LIN {X 0,Y 516.781,Z 239.858,A -85,B 0,C 180,E1 -4940.608,E2 -4940.608} C_VEL
LIN {X 0,Y 516.85,Z 239.104,A -85,B 0,C 180,E1 -4941.398,E2 -4941.398} C_VEL
LIN {X 0,Y 517,Z 239.087,A -85,B 0,C 180,E1 -4943.757,E2 -4943.757} C_VEL
LIN {X 0,Y 517.072,Z 239.077,A -85,B 0,C 180,E1 -4947.663,E2 -4947.663} C_VEL
LIN {X 0,Y 517.085,Z 239.079,A -85,B 0,C 180,E1 -4950.779,E2 -4950.779} C_VEL
LIN {X 0,Y 517.006,Z 239.087,A -85,B 0,C 180,E1 -4953.117,E2 -4953.117} C_VEL
LIN {X 0,Y 517,Z 239.087,A -85,B 0,C 180,E1 -4956.243,E2 -4956.243} C_VEL
LIN {X 0,Y 516.949,Z 239.094,A -85,B 0,C 180,E1 -4959.389,E2 -4959.389} C_VEL
LIN {X 0,Y 516.972,Z 239.092,A -85,B 0,C 180,E1 -4961.824,E2 -4961.824} C_VEL
LIN {X 0,Y 516.933,Z 239.096,A -85,B 0,C 180,E1 -4965.147,E2 -4965.147} C_VEL
LIN {X 0,Y 516.915,Z 239.097,A -85,B 0,C 180,E1 -4968.222,E2 -4968.222} C_VEL
LIN {X 0,Y 516.904,Z 239.098,A -85,B 0,C 180,E1 -4970.702,E2 -4970.702} C_VEL
LIN {X 0,Y 516.881,Z 239.1,A -85,B 0,C 180,E1 -4973.223,E2 -4973.223} C_VEL
LIN {X 0,Y 516.934,Z 239.096,A -85,B 0,C 180,E1 -4976.197,E2 -4976.197} C_VEL
LIN {X 0,Y 516.925,Z 239.096,A -85,B 0,C 180,E1 -4979.304,E2 -4979.304} C_VEL
LIN {X 0,Y 516.889,Z 239.099,A -85,B 0,C 180,E1 -4982.545,E2 -4982.545} C_VEL
LIN {X 0,Y 516.871,Z 239.103,A -85,B 0,C 180,E1 -4985.333,E2 -4985.333} C_VEL
LIN {X 0,Y 516.871,Z 239.105,A -85,B 0,C 180,E1 -4987.944,E2 -4987.944} C_VEL
LIN {X 0,Y 516.893,Z 239.1,A -85,B 0,C 180,E1 -4990.74,E2 -4990.74} C_VEL
LIN {X 0,Y 516.872,Z 239.105,A -85,B 0,C 180,E1 -4993.903,E2 -4993.903} C_VEL
LIN {X 0,Y 516.872,Z 239.103,A -85,B 0,C 180,E1 -4996.107,E2 -4996.107} C_VEL
LIN {X 0,Y 516.893,Z 239.1,A -85,B 0,C 180,E1 -4999.261,E2 -4999.261} C_VEL
LIN {X 0,Y 516.871,Z 239.103,A -85,B 0,C 180,E1 -5002.057,E2 -5002.057} C_VEL
LIN {X 0,Y 516.884,Z 239.102,A -85,B 0,C 180,E1 -5005.177,E2 -5005.177} C_VEL
LIN {X 0,Y 516.872,Z 239.102,A -85,B 0,C 180,E1 -5007.976,E2 -5007.976} C_VEL
LIN {X 0,Y 516.926,Z 239.097,A -85,B 0,C 180,E1 -5010.697,E2 -5010.697} C_VEL
LIN {X 0,Y 516.935,Z 239.093,A -85,B 0,C 180,E1 -5013.804,E2 -5013.804} C_VEL
LIN {X 0,Y 516.862,Z 239.106,A -85,B 0,C 180,E1 -5016.777,E2 -5016.777} C_VEL
LIN {X 0,Y 516.93,Z 239.094,A -85,B 0,C 180,E1 -5019.732,E2 -5019.732} C_VEL
LIN {X 0,Y 516.922,Z 239.097,A -85,B 0,C 180,E1 -5022.597,E2 -5022.597} C_VEL
LIN {X 0,Y 516.933,Z 239.097,A -85,B 0,C 180,E1 -5025.031,E2 -5025.031} C_VEL
LIN {X 0,Y 516.957,Z 239.092,A -85,B 0,C 180,E1 -5028.235,E2 -5028.235} C_VEL
LIN {X 0,Y 516.964,Z 239.092,A -85,B 0,C 180,E1 -5031.401,E2 -5031.401} C_VEL
LIN {X 0,Y 517.002,Z 239.088,A -85,B 0,C 180,E1 -5033.758,E2 -5033.758} C_VEL
LIN {X 0,Y 517.077,Z 239.077,A -85,B 0,C 180,E1 -5037.664,E2 -5037.664} C_VEL
LIN {X 0,Y 517.089,Z 239.077,A -85,B 0,C 180,E1 -5040.78,E2 -5040.78} C_VEL
LIN {X 0,Y 517.008,Z 239.086,A -85,B 0,C 180,E1 -5043.118,E2 -5043.118} C_VEL
LIN {X 0,Y 517.003,Z 239.086,A -85,B 0,C 180,E1 -5046.244,E2 -5046.244} C_VEL
LIN {X 0,Y 516.947,Z 239.095,A -85,B 0,C 180,E1 -5049.39,E2 -5049.39} C_VEL
LIN {X 0,Y 516.978,Z 239.091,A -85,B 0,C 180,E1 -5051.825,E2 -5051.825} C_VEL
LIN {X 0,Y 516.939,Z 239.095,A -85,B 0,C 180,E1 -5055.147,E2 -5055.147} C_VEL
LIN {X 0,Y 516.921,Z 239.096,A -85,B 0,C 180,E1 -5058.223,E2 -5058.223} C_VEL
LIN {X 0,Y 516.908,Z 239.097,A -85,B 0,C 180,E1 -5060.702,E2 -5060.702} C_VEL
LIN {X 0,Y 516.908,Z 239.098,A -85,B 0,C 180,E1 -5064.073,E2 -5064.073} C_VEL
LIN {X 0,Y 516.923,Z 239.095,A -85,B 0,C 180,E1 -5066.659,E2 -5066.659} C_VEL
LIN {X 0,Y 516.908,Z 239.1,A -85,B 0,C 180,E1 -5069.525,E2 -5069.525} C_VEL
LIN {X 0,Y 516.891,Z 239.099,A -85,B 0,C 180,E1 -5072.544,E2 -5072.544} C_VEL
LIN {X 0,Y 516.878,Z 239.103,A -85,B 0,C 180,E1 -5075.333,E2 -5075.333} C_VEL
LIN {X 0,Y 516.88,Z 239.103,A -85,B 0,C 180,E1 -5077.944,E2 -5077.944} C_VEL
LIN {X 0,Y 516.883,Z 239.102,A -85,B 0,C 180,E1 -5080.742,E2 -5080.742} C_VEL
LIN {X 0,Y 516.882,Z 239.103,A -85,B 0,C 180,E1 -5082.832,E2 -5082.832} C_VEL
LIN {X 0,Y 516.895,Z 239.101,A -85,B 0,C 180,E1 -5085.008,E2 -5085.008} C_VEL
LIN {X 0,Y 516.917,Z 239.097,A -85,B 0,C 180,E1 -5088.399,E2 -5088.399} C_VEL
LIN {X 0,Y 516.883,Z 239.102,A -85,B 0,C 180,E1 -5091.285,E2 -5091.285} C_VEL
LIN {X 0,Y 516.887,Z 239.123,A -85,B 0,C 180,E1 -5092.277,E2 -5092.277} C_VEL
LIN {X 0,Y 517.553,Z 243.494,A -85,B 0,C 180,E1 -5094.275,E2 -5094.275} C_VEL
LIN {X 0,Y 517.476,Z 248.974,A -85,B 0,C 180,E1 -5096.631,E2 -5096.631} C_VEL
LIN {X 0,Y 517.259,Z 255.571,A -85,B 0,C 180,E1 -5099.369,E2 -5099.369} C_VEL
LIN {X 0,Y 517.082,Z 262.252,A -85,B 0,C 180,E1 -5102.063,E2 -5102.063} C_VEL
LIN {X 0,Y 516.871,Z 269.94,A -85,B 0,C 180,E1 -5105.07,E2 -5105.07} C_VEL
LIN {X 0,Y 516.754,Z 277.811,A -85,B 0,C 180,E1 -5108.046,E2 -5108.046} C_VEL
LIN {X 0,Y 516.65,Z 285.647,A -85,B 0,C 180,E1 -5110.945,E2 -5110.945} C_VEL
LIN {X 0,Y 516.556,Z 294.588,A -85,B 0,C 180,E1 -5114.21,E2 -5114.21} C_VEL
LIN {X 0,Y 516.475,Z 299.805,A -85,B 0,C 180,E1 -5116.098,E2 -5116.098} C_VEL
LIN {X 0,Y 518.444,Z 312.994,A -85,B 0,C 180,E1 -5116.477,E2 -5116.477} C_VEL
LIN {X 0,Y 518.159,Z 326.349,A -85,B 0,C 180,E1 -5116.968,E2 -5116.968} C_VEL
LIN {X 0,Y 517.84,Z 339.017,A -85,B 0,C 180,E1 -5117.611,E2 -5117.611} C_VEL
LIN {X 0,Y 517.528,Z 350.117,A -85,B 0,C 180,E1 -5118.346,E2 -5118.346} C_VEL
LIN {X 0,Y 517.27,Z 360.807,A -85,B 0,C 180,E1 -5119.233,E2 -5119.233} C_VEL
LIN {X 0,Y 516.954,Z 370.437,A -85,B 0,C 180,E1 -5120.216,E2 -5120.216} C_VEL
LIN {X 0,Y 516.748,Z 378.335,A -85,B 0,C 180,E1 -5121.199,E2 -5121.199} C_VEL
LIN {X 0,Y 516.557,Z 386.049,A -85,B 0,C 180,E1 -5122.377,E2 -5122.377} C_VEL
LIN {X 0,Y 516.41,Z 393.155,A -85,B 0,C 180,E1 -5123.75,E2 -5123.75} C_VEL
LIN {X 0,Y 516.313,Z 397.881,A -85,B 0,C 180,E1 -5124.924,E2 -5124.924} C_VEL
LIN {X 0,Y 516.353,Z 401.495,A -85,B 0,C 180,E1 -5126.098,E2 -5126.098} C_VEL
LIN {X 0,Y 516.283,Z 403.356,A -85,B 0,C 180,E1 -5126.879,E2 -5126.879} C_VEL
LIN {X 0,Y 516.262,Z 404.752,A -85,B 0,C 180,E1 -5127.659,E2 -5127.659} C_VEL
LIN {X 0,Y 516.16,Z 406.353,A -85,B 0,C 180,E1 -5129.22,E2 -5129.22} C_VEL
LIN {X 0,Y 516.154,Z 406.567,A -85,B 0,C 180,E1 -5130,E2 -5130} C_VEL
LIN {X 0,Y 516.192,Z 405.742,A -85,B 0,C 180,E1 -5131.56,E2 -5131.56} C_VEL
LIN {X 0,Y 516.262,Z 404.747,A -85,B 0,C 180,E1 -5132.34,E2 -5132.34} C_VEL
LIN {X 0,Y 516.283,Z 403.347,A -85,B 0,C 180,E1 -5133.121,E2 -5133.121} C_VEL
LIN {X 0,Y 516.312,Z 400.405,A -85,B 0,C 180,E1 -5134.293,E2 -5134.293} C_VEL
LIN {X 0,Y 516.376,Z 396.423,A -85,B 0,C 180,E1 -5135.467,E2 -5135.467} C_VEL
LIN {X 0,Y 516.476,Z 390.537,A -85,B 0,C 180,E1 -5136.792,E2 -5136.792} C_VEL
LIN {X 0,Y 516.607,Z 383.603,A -85,B 0,C 180,E1 -5138.015,E2 -5138.015} C_VEL
LIN {X 0,Y 516.828,Z 375.295,A -85,B 0,C 180,E1 -5139.194,E2 -5139.194} C_VEL
LIN {X 0,Y 517.045,Z 366.775,A -85,B 0,C 180,E1 -5140.178,E2 -5140.178} C_VEL
LIN {X 0,Y 517.372,Z 356.252,A -85,B 0,C 180,E1 -5141.161,E2 -5141.161} C_VEL
LIN {X 0,Y 517.64,Z 345.343,A -85,B 0,C 180,E1 -5141.984,E2 -5141.984} C_VEL
LIN {X 0,Y 517.922,Z 334.436,A -85,B 0,C 180,E1 -5142.639,E2 -5142.639} C_VEL
LIN {X 0,Y 518.242,Z 322.713,A -85,B 0,C 180,E1 -5143.179,E2 -5143.179} C_VEL
LIN {X 0,Y 518.222,Z 311.055,A -85,B 0,C 180,E1 -5143.579,E2 -5143.579} C_VEL
LIN {X 0,Y 516.474,Z 299.644,A -85,B 0,C 180,E1 -5143.901,E2 -5143.901} C_VEL
LIN {X 0,Y 516.546,Z 290.986,A -85,B 0,C 180,E1 -5147.009,E2 -5147.009} C_VEL
LIN {X 0,Y 516.662,Z 282.256,A -85,B 0,C 180,E1 -5150.183,E2 -5150.183} C_VEL
LIN {X 0,Y 516.778,Z 274.076,A -85,B 0,C 180,E1 -5153.227,E2 -5153.227} C_VEL
LIN {X 0,Y 516.93,Z 266.37,A -85,B 0,C 180,E1 -5156.192,E2 -5156.192} C_VEL
LIN {X 0,Y 517.175,Z 257.911,A -85,B 0,C 180,E1 -5159.574,E2 -5159.574} C_VEL
LIN {X 0,Y 517.338,Z 252.096,A -85,B 0,C 180,E1 -5161.992,E2 -5161.992} C_VEL
LIN {X 0,Y 517.55,Z 245.678,A -85,B 0,C 180,E1 -5164.773,E2 -5164.773} C_VEL
LIN {X 0,Y 517.485,Z 242.522,A -85,B 0,C 180,E1 -5166.211,E2 -5166.211} C_VEL
LIN {X 0,Y 516.903,Z 239.1,A -85,B 0,C 180,E1 -5167.945,E2 -5167.945} C_VEL
LIN {X 0,Y 516.883,Z 239.103,A -85,B 0,C 180,E1 -5170.741,E2 -5170.741} C_VEL
LIN {X 0,Y 516.904,Z 239.099,A -85,B 0,C 180,E1 -5172.828,E2 -5172.828} C_VEL
LIN {X 0,Y 516.921,Z 239.097,A -85,B 0,C 180,E1 -5175.009,E2 -5175.009} C_VEL
LIN {X 0,Y 516.921,Z 239.099,A -85,B 0,C 180,E1 -5178.397,E2 -5178.397} C_VEL
LIN {X 0,Y 516.884,Z 239.103,A -85,B 0,C 180,E1 -5181.284,E2 -5181.284} C_VEL
LIN {X 0,Y 516.889,Z 239.101,A -85,B 0,C 180,E1 -5184.22,E2 -5184.22} C_VEL
LIN {X 0,Y 516.894,Z 239.101,A -85,B 0,C 180,E1 -5187.052,E2 -5187.052} C_VEL
LIN {X 0,Y 516.898,Z 239.101,A -85,B 0,C 180,E1 -5189.796,E2 -5189.796} C_VEL
LIN {X 0,Y 516.924,Z 239.096,A -85,B 0,C 180,E1 -5192.466,E2 -5192.466} C_VEL
LIN {X 0,Y 516.905,Z 239.1,A -85,B 0,C 180,E1 -5195.071,E2 -5195.071} C_VEL
LIN {X 0,Y 516.864,Z 239.104,A -85,B 0,C 180,E1 -5197.621,E2 -5197.621} C_VEL
LIN {X 0,Y 516.926,Z 239.098,A -85,B 0,C 180,E1 -5200.129,E2 -5200.129} C_VEL
LIN {X 0,Y 516.925,Z 239.096,A -85,B 0,C 180,E1 -5202.595,E2 -5202.595} C_VEL
LIN {X 0,Y 516.935,Z 239.096,A -85,B 0,C 180,E1 -5205.029,E2 -5205.029} C_VEL
LIN {X 0,Y 516.958,Z 239.094,A -85,B 0,C 180,E1 -5208.233,E2 -5208.233} C_VEL
LIN {X 0,Y 516.966,Z 239.093,A -85,B 0,C 180,E1 -5211.399,E2 -5211.399} C_VEL
LIN {X 0,Y 517.003,Z 239.087,A -85,B 0,C 180,E1 -5213.756,E2 -5213.756} C_VEL
LIN {X 0,Y 517.008,Z 239.086,A -85,B 0,C 180,E1 -5216.882,E2 -5216.882} C_VEL
LIN {X 0,Y 517.076,Z 239.078,A -85,B 0,C 180,E1 -5219.999,E2 -5219.999} C_VEL
LIN {X 0,Y 517.009,Z 239.087,A -85,B 0,C 180,E1 -5223.116,E2 -5223.116} C_VEL
LIN {X 0,Y 517.002,Z 239.087,A -85,B 0,C 180,E1 -5226.242,E2 -5226.242} C_VEL
LIN {X 0,Y 516.938,Z 239.096,A -85,B 0,C 180,E1 -5229.388,E2 -5229.388} C_VEL
LIN {X 0,Y 516.852,Z 239.109,A -85,B 0,C 180,E1 -5230.181,E2 -5230.181} C_VEL
LIN {X 0,Y 516.871,Z 239.697,A -85,B 0,C 180,E1 -5230.973,E2 -5230.973} C_VEL
LIN {X 0,Y 516.812,Z 243.273,A -85,B 0,C 180,E1 -5233.365,E2 -5233.365} C_VEL
LIN {X 0,Y 516.772,Z 246.951,A -85,B 0,C 180,E1 -5235.782,E2 -5235.782} C_VEL
LIN {X 0,Y 516.66,Z 250.764,A -85,B 0,C 180,E1 -5238.231,E2 -5238.231} C_VEL
LIN {X 0,Y 516.602,Z 254.676,A -85,B 0,C 180,E1 -5240.713,E2 -5240.713} C_VEL
LIN {X 0,Y 516.512,Z 258.727,A -85,B 0,C 180,E1 -5243.239,E2 -5243.239} C_VEL
LIN {X 0,Y 516.464,Z 263.377,A -85,B 0,C 180,E1 -5246.09,E2 -5246.09} C_VEL
LIN {X 0,Y 516.368,Z 267.257,A -85,B 0,C 180,E1 -5248.447,E2 -5248.447} C_VEL
LIN {X 0,Y 516.307,Z 271.751,A -85,B 0,C 180,E1 -5251.147,E2 -5251.147} C_VEL
LIN {X 0,Y 516.332,Z 273.494,A -85,B 0,C 180,E1 -5252.181,E2 -5252.181} C_VEL
LIN {X 0,Y 518.441,Z 284.959,A -85,B 0,C 180,E1 -5252.535,E2 -5252.535} C_VEL
LIN {X 0,Y 518.197,Z 298.137,A -85,B 0,C 180,E1 -5253.026,E2 -5253.026} C_VEL
LIN {X 0,Y 517.923,Z 309.971,A -85,B 0,C 180,E1 -5253.627,E2 -5253.627} C_VEL
LIN {X 0,Y 517.63,Z 321.625,A -85,B 0,C 180,E1 -5254.398,E2 -5254.398} C_VEL
LIN {X 0,Y 517.328,Z 331.516,A -85,B 0,C 180,E1 -5255.217,E2 -5255.217} C_VEL
LIN {X 0,Y 517.051,Z 341.592,A -85,B 0,C 180,E1 -5256.246,E2 -5256.246} C_VEL
LIN {X 0,Y 516.815,Z 349.52,A -85,B 0,C 180,E1 -5257.237,E2 -5257.237} C_VEL
LIN {X 0,Y 516.593,Z 357.769,A -85,B 0,C 180,E1 -5258.519,E2 -5258.519} C_VEL
LIN {X 0,Y 516.449,Z 364.091,A -85,B 0,C 180,E1 -5259.76,E2 -5259.76} C_VEL
LIN {X 0,Y 516.345,Z 369.595,A -85,B 0,C 180,E1 -5261.16,E2 -5261.16} C_VEL
LIN {X 0,Y 516.273,Z 372.805,A -85,B 0,C 180,E1 -5262.254,E2 -5262.254} C_VEL
LIN {X 0,Y 516.175,Z 375.193,A -85,B 0,C 180,E1 -5263.418,E2 -5263.418} C_VEL
LIN {X 0,Y 515.501,Z 376.253,A -85,B 0,C 180,E1 -5264.06,E2 -5264.06} C_VEL
LIN {X 0,Y 512.613,Z 377.313,A -85,B 0,C 180,E1 -5265.11,E2 -5265.11} C_VEL
LIN {X 0,Y 510.18,Z 377.672,A -85,B 0,C 180,E1 -5265.961,E2 -5265.961} C_VEL
LIN {X 0,Y 509.086,Z 377.559,A -85,B 0,C 180,E1 -5266.731,E2 -5266.731} C_VEL
LIN {X 0,Y 509.067,Z 377.457,A -85,B 0,C 180,E1 -5266.842,E2 -5266.842} C_VEL
LIN {X 0,Y 509.1,Z 376.219,A -85,B 0,C 180,E1 -5268.196,E2 -5268.196} C_VEL
LIN {X 0,Y 509.152,Z 373.756,A -85,B 0,C 180,E1 -5269.553,E2 -5269.553} C_VEL
LIN {X 0,Y 509.246,Z 369.376,A -85,B 0,C 180,E1 -5271.112,E2 -5271.112} C_VEL
LIN {X 0,Y 509.371,Z 365.032,A -85,B 0,C 180,E1 -5272.243,E2 -5272.243} C_VEL
LIN {X 0,Y 509.524,Z 358.201,A -85,B 0,C 180,E1 -5273.623,E2 -5273.623} C_VEL
LIN {X 0,Y 509.749,Z 350.466,A -85,B 0,C 180,E1 -5274.858,E2 -5274.858} C_VEL
LIN {X 0,Y 510.002,Z 342.168,A -85,B 0,C 180,E1 -5275.928,E2 -5275.928} C_VEL
LIN {X 0,Y 510.286,Z 333.086,A -85,B 0,C 180,E1 -5276.885,E2 -5276.885} C_VEL
LIN {X 0,Y 510.534,Z 322.887,A -85,B 0,C 180,E1 -5277.763,E2 -5277.763} C_VEL
LIN {X 0,Y 510.843,Z 311.745,A -85,B 0,C 180,E1 -5278.534,E2 -5278.534} C_VEL
LIN {X 0,Y 511.18,Z 300.598,A -85,B 0,C 180,E1 -5279.137,E2 -5279.137} C_VEL
LIN {X 0,Y 511.527,Z 287.847,A -85,B 0,C 180,E1 -5279.646,E2 -5279.646} C_VEL
LIN {X 0,Y 511.045,Z 282.976,A -85,B 0,C 180,E1 -5279.814,E2 -5279.814} C_VEL
LIN {X 0,Y 509.176,Z 273.536,A -85,B 0,C 180,E1 -5280.12,E2 -5280.12} C_VEL
LIN {X 0,Y 509.257,Z 268.829,A -85,B 0,C 180,E1 -5282.909,E2 -5282.909} C_VEL
LIN {X 0,Y 509.302,Z 264.37,A -85,B 0,C 180,E1 -5285.606,E2 -5285.606} C_VEL
LIN {X 0,Y 509.405,Z 260.256,A -85,B 0,C 180,E1 -5288.13,E2 -5288.13} C_VEL
LIN {X 0,Y 509.488,Z 256.157,A -85,B 0,C 180,E1 -5290.667,E2 -5290.667} C_VEL
LIN {X 0,Y 509.517,Z 252.195,A -85,B 0,C 180,E1 -5293.163,E2 -5293.163} C_VEL
LIN {X 0,Y 509.625,Z 248.325,A -85,B 0,C 180,E1 -5295.628,E2 -5295.628} C_VEL
LIN {X 0,Y 509.795,Z 243.32,A -85,B 0,C 180,E1 -5298.872,E2 -5298.872} C_VEL
LIN {X 0,Y 509.787,Z 239.984,A -85,B 0,C 180,E1 -5301.278,E2 -5301.278} C_VEL
LIN {X 0,Y 509.968,Z 239.963,A -85,B 0,C 180,E1 -5303.671,E2 -5303.671} C_VEL
LIN {X 0,Y 510.044,Z 239.952,A -85,B 0,C 180,E1 -5307.631,E2 -5307.631} C_VEL
LIN {X 0,Y 510.044,Z 239.953,A -85,B 0,C 180,E1 -5310,E2 -5310} C_VEL
LIN {X 0,Y 510.047,Z 239.953,A -85,B 0,C 180,E1 -5312.369,E2 -5312.369} C_VEL
LIN {X 0,Y 509.968,Z 239.963,A -85,B 0,C 180,E1 -5316.33,E2 -5316.33} C_VEL
LIN {X 0,Y 509.909,Z 239.97,A -85,B 0,C 180,E1 -5318.72,E2 -5318.72} C_VEL
LIN {X 0,Y 509.94,Z 239.967,A -85,B 0,C 180,E1 -5321.931,E2 -5321.931} C_VEL
LIN {X 0,Y 509.882,Z 239.974,A -85,B 0,C 180,E1 -5325.242,E2 -5325.242} C_VEL
LIN {X 0,Y 509.878,Z 239.974,A -85,B 0,C 180,E1 -5328.001,E2 -5328.001} C_VEL
LIN {X 0,Y 509.847,Z 239.978,A -85,B 0,C 180,E1 -5331.002,E2 -5331.002} C_VEL
LIN {X 0,Y 509.84,Z 239.98,A -85,B 0,C 180,E1 -5333.563,E2 -5333.563} C_VEL
LIN {X 0,Y 509.903,Z 239.97,A -85,B 0,C 180,E1 -5336.379,E2 -5336.379} C_VEL
LIN {X 0,Y 509.875,Z 239.973,A -85,B 0,C 180,E1 -5338.844,E2 -5338.844} C_VEL
LIN {X 0,Y 509.815,Z 239.982,A -85,B 0,C 180,E1 -5341.59,E2 -5341.59} C_VEL
LIN {X 0,Y 509.842,Z 239.979,A -85,B 0,C 180,E1 -5344.414,E2 -5344.414} C_VEL
LIN {X 0,Y 509.808,Z 239.983,A -85,B 0,C 180,E1 -5347.341,E2 -5347.341} C_VEL
LIN {X 0,Y 509.85,Z 239.978,A -85,B 0,C 180,E1 -5350.38,E2 -5350.38} C_VEL
LIN {X 0,Y 509.829,Z 239.981,A -85,B 0,C 180,E1 -5353.065,E2 -5353.065} C_VEL
LIN {X 0,Y 509.819,Z 239.981,A -85,B 0,C 180,E1 -5355.793,E2 -5355.793} C_VEL
LIN {X 0,Y 509.855,Z 239.976,A -85,B 0,C 180,E1 -5358.576,E2 -5358.576} C_VEL
LIN {X 0,Y 509.845,Z 239.977,A -85,B 0,C 180,E1 -5361.786,E2 -5361.786} C_VEL
LIN {X 0,Y 509.835,Z 239.979,A -85,B 0,C 180,E1 -5364.624,E2 -5364.624} C_VEL
LIN {X 0,Y 509.855,Z 239.977,A -85,B 0,C 180,E1 -5367.482,E2 -5367.482} C_VEL
LIN {X 0,Y 509.871,Z 239.973,A -85,B 0,C 180,E1 -5370.27,E2 -5370.27} C_VEL
LIN {X 0,Y 509.877,Z 239.975,A -85,B 0,C 180,E1 -5372.945,E2 -5372.945} C_VEL
LIN {X 0,Y 509.86,Z 239.977,A -85,B 0,C 180,E1 -5375.575,E2 -5375.575} C_VEL
LIN {X 0,Y 509.813,Z 239.983,A -85,B 0,C 180,E1 -5378.149,E2 -5378.149} C_VEL
LIN {X 0,Y 509.856,Z 239.978,A -85,B 0,C 180,E1 -5380.682,E2 -5380.682} C_VEL
LIN {X 0,Y 509.878,Z 239.973,A -85,B 0,C 180,E1 -5383.176,E2 -5383.176} C_VEL
LIN {X 0,Y 509.854,Z 239.976,A -85,B 0,C 180,E1 -5385.635,E2 -5385.635} C_VEL
LIN {X 0,Y 509.91,Z 239.971,A -85,B 0,C 180,E1 -5388.876,E2 -5388.876} C_VEL
LIN {X 0,Y 509.944,Z 239.965,A -85,B 0,C 180,E1 -5392.079,E2 -5392.079} C_VEL
LIN {X 0,Y 509.975,Z 239.962,A -85,B 0,C 180,E1 -5394.465,E2 -5394.465} C_VEL
LIN {X 0,Y 510.048,Z 239.953,A -85,B 0,C 180,E1 -5397.632,E2 -5397.632} C_VEL
LIN {X 0,Y 510.059,Z 239.952,A -85,B 0,C 180,E1 -5400.79,E2 -5400.79} C_VEL
LIN {X 0,Y 509.951,Z 239.965,A -85,B 0,C 180,E1 -5403.161,E2 -5403.161} C_VEL
LIN {X 0,Y 509.972,Z 239.962,A -85,B 0,C 180,E1 -5406.331,E2 -5406.331} C_VEL
LIN {X 0,Y 509.91,Z 239.969,A -85,B 0,C 180,E1 -5408.721,E2 -5408.721} C_VEL
LIN {X 0,Y 509.946,Z 239.966,A -85,B 0,C 180,E1 -5411.931,E2 -5411.931} C_VEL
LIN {X 0,Y 509.889,Z 239.974,A -85,B 0,C 180,E1 -5415.243,E2 -5415.243} C_VEL
LIN {X 0,Y 509.884,Z 239.973,A -85,B 0,C 180,E1 -5418.002,E2 -5418.002} C_VEL
LIN {X 0,Y 509.846,Z 239.977,A -85,B 0,C 180,E1 -5421.003,E2 -5421.003} C_VEL
LIN {X 0,Y 509.866,Z 239.975,A -85,B 0,C 180,E1 -5424.427,E2 -5424.427} C_VEL
LIN {X 0,Y 509.883,Z 239.973,A -85,B 0,C 180,E1 -5427.057,E2 -5427.057} C_VEL
LIN {X 0,Y 509.854,Z 239.978,A -85,B 0,C 180,E1 -5429.752,E2 -5429.752} C_VEL
LIN {X 0,Y 509.864,Z 239.975,A -85,B 0,C 180,E1 -5432.774,E2 -5432.774} C_VEL
LIN {X 0,Y 509.838,Z 239.981,A -85,B 0,C 180,E1 -5435.582,E2 -5435.582} C_VEL
LIN {X 0,Y 509.849,Z 239.977,A -85,B 0,C 180,E1 -5438.339,E2 -5438.339} C_VEL
LIN {X 0,Y 509.855,Z 239.978,A -85,B 0,C 180,E1 -5441.426,E2 -5441.426} C_VEL
LIN {X 0,Y 509.838,Z 239.978,A -85,B 0,C 180,E1 -5444.671,E2 -5444.671} C_VEL
LIN {X 0,Y 509.859,Z 239.976,A -85,B 0,C 180,E1 -5448.104,E2 -5448.104} C_VEL
LIN {X 0,Y 509.847,Z 239.977,A -85,B 0,C 180,E1 -5450.648,E2 -5450.648} C_VEL
LIN {X 0,Y 509.89,Z 240.142,A -85,B 0,C 180,E1 -5452.168,E2 -5452.168} C_VEL
LIN {X 0,Y 510.554,Z 244.774,A -85,B 0,C 180,E1 -5454.308,E2 -5454.308} C_VEL
LIN {X 0,Y 510.466,Z 250.003,A -85,B 0,C 180,E1 -5456.585,E2 -5456.585} C_VEL
LIN {X 0,Y 510.23,Z 256.59,A -85,B 0,C 180,E1 -5459.36,E2 -5459.36} C_VEL
LIN {X 0,Y 510.045,Z 263.199,A -85,B 0,C 180,E1 -5462.064,E2 -5462.064} C_VEL
LIN {X 0,Y 509.856,Z 269.825,A -85,B 0,C 180,E1 -5464.703,E2 -5464.703} C_VEL
LIN {X 0,Y 509.723,Z 277.003,A -85,B 0,C 180,E1 -5467.487,E2 -5467.487} C_VEL
LIN {X 0,Y 509.588,Z 285.451,A -85,B 0,C 180,E1 -5470.671,E2 -5470.671} C_VEL
LIN {X 0,Y 509.484,Z 294.395,A -85,B 0,C 180,E1 -5473.985,E2 -5473.985} C_VEL
LIN {X 0,Y 509.387,Z 299.615,A -85,B 0,C 180,E1 -5475.901,E2 -5475.901} C_VEL
LIN {X 0,Y 511.503,Z 313.527,A -85,B 0,C 180,E1 -5476.315,E2 -5476.315} C_VEL
LIN {X 0,Y 511.216,Z 326.109,A -85,B 0,C 180,E1 -5476.788,E2 -5476.788} C_VEL
LIN {X 0,Y 510.891,Z 338.842,A -85,B 0,C 180,E1 -5477.443,E2 -5477.443} C_VEL
LIN {X 0,Y 510.528,Z 349.891,A -85,B 0,C 180,E1 -5478.184,E2 -5478.184} C_VEL
LIN {X 0,Y 510.269,Z 360.585,A -85,B 0,C 180,E1 -5479.083,E2 -5479.083} C_VEL
LIN {X 0,Y 509.921,Z 370.219,A -85,B 0,C 180,E1 -5480.08,E2 -5480.08} C_VEL
LIN {X 0,Y 509.696,Z 378.122,A -85,B 0,C 180,E1 -5481.076,E2 -5481.076} C_VEL
LIN {X 0,Y 509.488,Z 385.841,A -85,B 0,C 180,E1 -5482.271,E2 -5482.271} C_VEL
LIN {X 0,Y 509.322,Z 392.077,A -85,B 0,C 180,E1 -5483.472,E2 -5483.472} C_VEL
LIN {X 0,Y 509.244,Z 397.679,A -85,B 0,C 180,E1 -5484.853,E2 -5484.853} C_VEL
LIN {X 0,Y 509.246,Z 401.294,A -85,B 0,C 180,E1 -5486.043,E2 -5486.043} C_VEL
LIN {X 0,Y 509.201,Z 403.157,A -85,B 0,C 180,E1 -5486.835,E2 -5486.835} C_VEL
LIN {X 0,Y 509.19,Z 404.554,A -85,B 0,C 180,E1 -5487.627,E2 -5487.627} C_VEL
LIN {X 0,Y 509.074,Z 406.154,A -85,B 0,C 180,E1 -5489.209,E2 -5489.209} C_VEL
LIN {X 0,Y 509.066,Z 406.368,A -85,B 0,C 180,E1 -5490,E2 -5490} C_VEL
LIN {X 0,Y 509.113,Z 405.541,A -85,B 0,C 180,E1 -5491.582,E2 -5491.582} C_VEL
LIN {X 0,Y 509.19,Z 404.543,A -85,B 0,C 180,E1 -5492.373,E2 -5492.373} C_VEL
LIN {X 0,Y 509.201,Z 403.142,A -85,B 0,C 180,E1 -5493.165,E2 -5493.165} C_VEL
LIN {X 0,Y 509.205,Z 400.196,A -85,B 0,C 180,E1 -5494.353,E2 -5494.353} C_VEL
LIN {X 0,Y 509.294,Z 396.21,A -85,B 0,C 180,E1 -5495.543,E2 -5495.543} C_VEL
LIN {X 0,Y 509.409,Z 390.179,A -85,B 0,C 180,E1 -5496.913,E2 -5496.913} C_VEL
LIN {X 0,Y 509.552,Z 383.376,A -85,B 0,C 180,E1 -5498.127,E2 -5498.127} C_VEL
LIN {X 0,Y 509.775,Z 375.061,A -85,B 0,C 180,E1 -5499.322,E2 -5499.322} C_VEL
LIN {X 0,Y 510.022,Z 366.533,A -85,B 0,C 180,E1 -5500.319,E2 -5500.319} C_VEL
LIN {X 0,Y 510.374,Z 356.002,A -85,B 0,C 180,E1 -5501.316,E2 -5501.316} C_VEL
LIN {X 0,Y 510.643,Z 345.085,A -85,B 0,C 180,E1 -5502.151,E2 -5502.151} C_VEL
LIN {X 0,Y 510.975,Z 334.171,A -85,B 0,C 180,E1 -5502.814,E2 -5502.814} C_VEL
LIN {X 0,Y 511.304,Z 322.434,A -85,B 0,C 180,E1 -5503.361,E2 -5503.361} C_VEL
LIN {X 0,Y 511.295,Z 311.683,A -85,B 0,C 180,E1 -5503.741,E2 -5503.741} C_VEL
LIN {X 0,Y 509.377,Z 299.421,A -85,B 0,C 180,E1 -5504.099,E2 -5504.099} C_VEL
LIN {X 0,Y 509.486,Z 290.761,A -85,B 0,C 180,E1 -5507.252,E2 -5507.252} C_VEL
LIN {X 0,Y 509.593,Z 282.525,A -85,B 0,C 180,E1 -5510.311,E2 -5510.311} C_VEL
LIN {X 0,Y 509.73,Z 275.073,A -85,B 0,C 180,E1 -5513.138,E2 -5513.138} C_VEL
LIN {X 0,Y 509.906,Z 266.783,A -85,B 0,C 180,E1 -5516.376,E2 -5516.376} C_VEL
LIN {X 0,Y 510.14,Z 258.414,A -85,B 0,C 180,E1 -5519.781,E2 -5519.781} C_VEL
LIN {X 0,Y 510.39,Z 251.18,A -85,B 0,C 180,E1 -5522.863,E2 -5522.863} C_VEL
LIN {X 0,Y 510.574,Z 244.858,A -85,B 0,C 180,E1 -5525.695,E2 -5525.695} C_VEL
LIN {X 0,Y 509.864,Z 239.978,A -85,B 0,C 180,E1 -5528.145,E2 -5528.145} C_VEL
LIN {X 0,Y 509.856,Z 239.979,A -85,B 0,C 180,E1 -5531.424,E2 -5531.424} C_VEL
LIN {X 0,Y 509.855,Z 239.978,A -85,B 0,C 180,E1 -5534.667,E2 -5534.667} C_VEL
LIN {X 0,Y 509.859,Z 239.977,A -85,B 0,C 180,E1 -5538.102,E2 -5538.102} C_VEL
LIN {X 0,Y 509.857,Z 239.98,A -85,B 0,C 180,E1 -5540.648,E2 -5540.648} C_VEL
LIN {X 0,Y 509.834,Z 239.982,A -85,B 0,C 180,E1 -5543.647,E2 -5543.647} C_VEL
LIN {X 0,Y 509.859,Z 239.978,A -85,B 0,C 180,E1 -5546.538,E2 -5546.538} C_VEL
LIN {X 0,Y 509.847,Z 239.978,A -85,B 0,C 180,E1 -5549.334,E2 -5549.334} C_VEL
LIN {X 0,Y 509.89,Z 239.973,A -85,B 0,C 180,E1 -5552.054,E2 -5552.054} C_VEL
LIN {X 0,Y 509.872,Z 239.976,A -85,B 0,C 180,E1 -5554.703,E2 -5554.703} C_VEL
LIN {X 0,Y 509.822,Z 239.981,A -85,B 0,C 180,E1 -5557.456,E2 -5557.456} C_VEL
LIN {X 0,Y 509.911,Z 239.971,A -85,B 0,C 180,E1 -5559.844,E2 -5559.844} C_VEL
LIN {X 0,Y 509.881,Z 239.976,A -85,B 0,C 180,E1 -5563.174,E2 -5563.174} C_VEL
LIN {X 0,Y 509.858,Z 239.977,A -85,B 0,C 180,E1 -5565.633,E2 -5565.633} C_VEL
LIN {X 0,Y 509.911,Z 239.97,A -85,B 0,C 180,E1 -5568.874,E2 -5568.874} C_VEL
LIN {X 0,Y 509.945,Z 239.966,A -85,B 0,C 180,E1 -5572.077,E2 -5572.077} C_VEL
LIN {X 0,Y 509.977,Z 239.963,A -85,B 0,C 180,E1 -5574.463,E2 -5574.463} C_VEL
LIN {X 0,Y 510.047,Z 239.955,A -85,B 0,C 180,E1 -5577.63,E2 -5577.63} C_VEL
LIN {X 0,Y 510.057,Z 239.953,A -85,B 0,C 180,E1 -5580.789,E2 -5580.789} C_VEL
LIN {X 0,Y 509.951,Z 239.966,A -85,B 0,C 180,E1 -5583.159,E2 -5583.159} C_VEL
LIN {X 0,Y 509.97,Z 239.963,A -85,B 0,C 180,E1 -5586.329,E2 -5586.329} C_VEL
LIN {X 0,Y 509.907,Z 239.973,A -85,B 0,C 180,E1 -5588.719,E2 -5588.719} C_VEL
LIN {X 0,Y 509.791,Z 239.989,A -85,B 0,C 180,E1 -5590.323,E2 -5590.323} C_VEL
LIN {X 0,Y 509.858,Z 242.042,A -85,B 0,C 180,E1 -5591.932,E2 -5591.932} C_VEL
LIN {X 0,Y 509.747,Z 246.901,A -85,B 0,C 180,E1 -5595.185,E2 -5595.185} C_VEL
LIN {X 0,Y 509.642,Z 251.084,A -85,B 0,C 180,E1 -5597.919,E2 -5597.919} C_VEL
LIN {X 0,Y 509.508,Z 255.884,A -85,B 0,C 180,E1 -5601.015,E2 -5601.015} C_VEL
LIN {X 0,Y 509.429,Z 259.988,A -85,B 0,C 180,E1 -5603.582,E2 -5603.582} C_VEL
LIN {X 0,Y 509.392,Z 264.302,A -85,B 0,C 180,E1 -5606.263,E2 -5606.263} C_VEL
LIN {X 0,Y 509.279,Z 268.575,A -85,B 0,C 180,E1 -5608.88,E2 -5608.88} C_VEL
LIN {X 0,Y 509.258,Z 273.702,A -85,B 0,C 180,E1 -5611.977,E2 -5611.977} C_VEL
LIN {X 0,Y 511.513,Z 286.226,A -85,B 0,C 180,E1 -5612.385,E2 -5612.385} C_VEL
LIN {X 0,Y 511.28,Z 298.858,A -85,B 0,C 180,E1 -5612.872,E2 -5612.872} C_VEL
LIN {X 0,Y 510.98,Z 310.801,A -85,B 0,C 180,E1 -5613.494,E2 -5613.494} C_VEL
LIN {X 0,Y 510.657,Z 322.087,A -85,B 0,C 180,E1 -5614.26,E2 -5614.26} C_VEL
LIN {X 0,Y 510.317,Z 333.282,A -85,B 0,C 180,E1 -5615.217,E2 -5615.217} C_VEL
LIN {X 0,Y 510.038,Z 342.078,A -85,B 0,C 180,E1 -5616.144,E2 -5616.144} C_VEL
LIN {X 0,Y 509.807,Z 349.558,A -85,B 0,C 180,E1 -5617.095,E2 -5617.095} C_VEL
LIN {X 0,Y 509.553,Z 357.672,A -85,B 0,C 180,E1 -5618.363,E2 -5618.363} C_VEL
LIN {X 0,Y 509.393,Z 364.178,A -85,B 0,C 180,E1 -5619.648,E2 -5619.648} C_VEL
LIN {X 0,Y 509.27,Z 369.573,A -85,B 0,C 180,E1 -5621.025,E2 -5621.025} C_VEL
LIN {X 0,Y 509.23,Z 371.983,A -85,B 0,C 180,E1 -5621.819,E2 -5621.819} C_VEL
LIN {X 0,Y 509.11,Z 374.729,A -85,B 0,C 180,E1 -5622.977,E2 -5622.977} C_VEL
LIN {X 0,Y 509.1,Z 376.556,A -85,B 0,C 180,E1 -5624.124,E2 -5624.124} C_VEL
LIN {X 0,Y 509.102,Z 377.498,A -85,B 0,C 180,E1 -5625.249,E2 -5625.249} C_VEL
LIN {X 0,Y 509.077,Z 377.658,A -85,B 0,C 180,E1 -5626.35,E2 -5626.35} C_VEL
LIN {X 0,Y 509.067,Z 377.457,A -85,B 0,C 180,E1 -5626.842,E2 -5626.842} C_VEL
LIN {X 0,Y 508.416,Z 377.061,A -85,B 0,C 180,E1 -5627.502,E2 -5627.502} C_VEL
LIN {X 0,Y 505.578,Z 375.823,A -85,B 0,C 180,E1 -5628.567,E2 -5628.567} C_VEL
LIN {X 0,Y 503.187,Z 374.316,A -85,B 0,C 180,E1 -5629.416,E2 -5629.416} C_VEL
LIN {X 0,Y 502.178,Z 372.853,A -85,B 0,C 180,E1 -5630.062,E2 -5630.062} C_VEL
LIN {X 0,Y 502.107,Z 372.281,A -85,B 0,C 180,E1 -5630.279,E2 -5630.279} C_VEL
LIN {X 0,Y 502.217,Z 368.114,A -85,B 0,C 180,E1 -5631.595,E2 -5631.595} C_VEL
LIN {X 0,Y 502.365,Z 362.072,A -85,B 0,C 180,E1 -5633.019,E2 -5633.019} C_VEL
LIN {X 0,Y 502.591,Z 354.402,A -85,B 0,C 180,E1 -5634.409,E2 -5634.409} C_VEL
LIN {X 0,Y 502.843,Z 346.536,A -85,B 0,C 180,E1 -5635.547,E2 -5635.547} C_VEL
LIN {X 0,Y 503.172,Z 337.297,A -85,B 0,C 180,E1 -5636.627,E2 -5636.627} C_VEL
LIN {X 0,Y 503.479,Z 326.916,A -85,B 0,C 180,E1 -5637.611,E2 -5637.611} C_VEL
LIN {X 0,Y 503.81,Z 316.676,A -85,B 0,C 180,E1 -5638.396,E2 -5638.396} C_VEL
LIN {X 0,Y 504.08,Z 305.816,A -85,B 0,C 180,E1 -5639.062,E2 -5639.062} C_VEL
LIN {X 0,Y 504.499,Z 293.122,A -85,B 0,C 180,E1 -5639.648,E2 -5639.648} C_VEL
LIN {X 0,Y 504.471,Z 285.768,A -85,B 0,C 180,E1 -5639.916,E2 -5639.916} C_VEL
LIN {X 0,Y 502.095,Z 273.703,A -85,B 0,C 180,E1 -5640.32,E2 -5640.32} C_VEL
LIN {X 0,Y 502.188,Z 268.596,A -85,B 0,C 180,E1 -5643.396,E2 -5643.396} C_VEL
LIN {X 0,Y 502.238,Z 264.247,A -85,B 0,C 180,E1 -5646.059,E2 -5646.059} C_VEL
LIN {X 0,Y 502.347,Z 260.031,A -85,B 0,C 180,E1 -5648.67,E2 -5648.67} C_VEL
LIN {X 0,Y 502.421,Z 255.955,A -85,B 0,C 180,E1 -5651.233,E2 -5651.233} C_VEL
LIN {X 0,Y 502.51,Z 250.7,A -85,B 0,C 180,E1 -5654.59,E2 -5654.59} C_VEL
LIN {X 0,Y 502.693,Z 245.617,A -85,B 0,C 180,E1 -5657.895,E2 -5657.895} C_VEL
LIN {X 0,Y 502.717,Z 240.866,A -85,B 0,C 180,E1 -5661.154,E2 -5661.154} C_VEL
LIN {X 0,Y 502.915,Z 240.842,A -85,B 0,C 180,E1 -5663.581,E2 -5663.581} C_VEL
LIN {X 0,Y 502.891,Z 240.845,A -85,B 0,C 180,E1 -5666.796,E2 -5666.796} C_VEL
LIN {X 0,Y 503.027,Z 240.827,A -85,B 0,C 180,E1 -5669.2,E2 -5669.2} C_VEL
LIN {X 0,Y 503.017,Z 240.829,A -85,B 0,C 180,E1 -5672.402,E2 -5672.402} C_VEL
LIN {X 0,Y 502.929,Z 240.84,A -85,B 0,C 180,E1 -5675.614,E2 -5675.614} C_VEL
LIN {X 0,Y 502.892,Z 240.846,A -85,B 0,C 180,E1 -5678.033,E2 -5678.033} C_VEL
LIN {X 0,Y 502.884,Z 240.844,A -85,B 0,C 180,E1 -5681.283,E2 -5681.283} C_VEL
LIN {X 0,Y 502.834,Z 240.851,A -85,B 0,C 180,E1 -5684.571,E2 -5684.571} C_VEL
LIN {X 0,Y 502.851,Z 240.85,A -85,B 0,C 180,E1 -5687.907,E2 -5687.907} C_VEL
LIN {X 0,Y 502.819,Z 240.852,A -85,B 0,C 180,E1 -5690.537,E2 -5690.537} C_VEL
LIN {X 0,Y 502.795,Z 240.854,A -85,B 0,C 180,E1 -5693.04,E2 -5693.04} C_VEL
LIN {X 0,Y 502.831,Z 240.852,A -85,B 0,C 180,E1 -5695.676,E2 -5695.676} C_VEL
LIN {X 0,Y 502.831,Z 240.853,A -85,B 0,C 180,E1 -5698.373,E2 -5698.373} C_VEL
LIN {X 0,Y 502.786,Z 240.857,A -85,B 0,C 180,E1 -5701.5,E2 -5701.5} C_VEL
LIN {X 0,Y 502.795,Z 240.857,A -85,B 0,C 180,E1 -5704.445,E2 -5704.445} C_VEL
LIN {X 0,Y 502.77,Z 240.86,A -85,B 0,C 180,E1 -5707.179,E2 -5707.179} C_VEL
LIN {X 0,Y 502.815,Z 240.854,A -85,B 0,C 180,E1 -5710.012,E2 -5710.012} C_VEL
LIN {X 0,Y 502.818,Z 240.852,A -85,B 0,C 180,E1 -5712.203,E2 -5712.203} C_VEL
LIN {X 0,Y 502.789,Z 240.858,A -85,B 0,C 180,E1 -5715.469,E2 -5715.469} C_VEL
LIN {X 0,Y 502.818,Z 240.853,A -85,B 0,C 180,E1 -5717.865,E2 -5717.865} C_VEL
LIN {X 0,Y 502.81,Z 240.855,A -85,B 0,C 180,E1 -5721.026,E2 -5721.026} C_VEL
LIN {X 0,Y 502.775,Z 240.857,A -85,B 0,C 180,E1 -5724.168,E2 -5724.168} C_VEL
LIN {X 0,Y 502.822,Z 240.854,A -85,B 0,C 180,E1 -5726.994,E2 -5726.994} C_VEL
LIN {X 0,Y 502.82,Z 240.852,A -85,B 0,C 180,E1 -5730.062,E2 -5730.062} C_VEL
LIN {X 0,Y 502.825,Z 240.852,A -85,B 0,C 180,E1 -5732.534,E2 -5732.534} C_VEL
LIN {X 0,Y 502.819,Z 240.854,A -85,B 0,C 180,E1 -5735.299,E2 -5735.299} C_VEL
LIN {X 0,Y 502.775,Z 240.859,A -85,B 0,C 180,E1 -5737.827,E2 -5737.827} C_VEL
LIN {X 0,Y 502.817,Z 240.855,A -85,B 0,C 180,E1 -5740.401,E2 -5740.401} C_VEL
LIN {X 0,Y 502.827,Z 240.853,A -85,B 0,C 180,E1 -5742.933,E2 -5742.933} C_VEL
LIN {X 0,Y 502.836,Z 240.851,A -85,B 0,C 180,E1 -5745.43,E2 -5745.43} C_VEL
LIN {X 0,Y 502.873,Z 240.849,A -85,B 0,C 180,E1 -5748.718,E2 -5748.718} C_VEL
LIN {X 0,Y 502.895,Z 240.843,A -85,B 0,C 180,E1 -5751.968,E2 -5751.968} C_VEL
LIN {X 0,Y 502.931,Z 240.839,A -85,B 0,C 180,E1 -5754.387,E2 -5754.387} C_VEL
LIN {X 0,Y 503.018,Z 240.828,A -85,B 0,C 180,E1 -5757.599,E2 -5757.599} C_VEL
LIN {X 0,Y 503.018,Z 240.829,A -85,B 0,C 180,E1 -5760.001,E2 -5760.001} C_VEL
LIN {X 0,Y 503.019,Z 240.828,A -85,B 0,C 180,E1 -5762.403,E2 -5762.403} C_VEL
LIN {X 0,Y 502.932,Z 240.84,A -85,B 0,C 180,E1 -5765.614,E2 -5765.614} C_VEL
LIN {X 0,Y 502.896,Z 240.846,A -85,B 0,C 180,E1 -5768.034,E2 -5768.034} C_VEL
LIN {X 0,Y 502.887,Z 240.843,A -85,B 0,C 180,E1 -5771.284,E2 -5771.284} C_VEL
LIN {X 0,Y 502.84,Z 240.849,A -85,B 0,C 180,E1 -5774.572,E2 -5774.572} C_VEL
LIN {X 0,Y 502.857,Z 240.849,A -85,B 0,C 180,E1 -5777.908,E2 -5777.908} C_VEL
LIN {X 0,Y 502.825,Z 240.851,A -85,B 0,C 180,E1 -5780.537,E2 -5780.537} C_VEL
LIN {X 0,Y 502.791,Z 240.856,A -85,B 0,C 180,E1 -5783.041,E2 -5783.041} C_VEL
LIN {X 0,Y 502.837,Z 240.852,A -85,B 0,C 180,E1 -5785.677,E2 -5785.677} C_VEL
LIN {X 0,Y 502.838,Z 240.851,A -85,B 0,C 180,E1 -5788.374,E2 -5788.374} C_VEL
LIN {X 0,Y 502.79,Z 240.857,A -85,B 0,C 180,E1 -5791.5,E2 -5791.5} C_VEL
LIN {X 0,Y 502.79,Z 240.857,A -85,B 0,C 180,E1 -5793.996,E2 -5793.996} C_VEL
LIN {X 0,Y 502.779,Z 240.859,A -85,B 0,C 180,E1 -5797.179,E2 -5797.179} C_VEL
LIN {X 0,Y 502.787,Z 240.857,A -85,B 0,C 180,E1 -5800.016,E2 -5800.016} C_VEL
LIN {X 0,Y 502.802,Z 240.853,A -85,B 0,C 180,E1 -5802.2,E2 -5802.2} C_VEL
LIN {X 0,Y 502.785,Z 240.857,A -85,B 0,C 180,E1 -5805.471,E2 -5805.471} C_VEL
LIN {X 0,Y 502.821,Z 240.854,A -85,B 0,C 180,E1 -5808.935,E2 -5808.935} C_VEL
LIN {X 0,Y 502.815,Z 240.872,A -85,B 0,C 180,E1 -5811.916,E2 -5811.916} C_VEL
LIN {X 0,Y 503.523,Z 245.535,A -85,B 0,C 180,E1 -5814.111,E2 -5814.111} C_VEL
LIN {X 0,Y 503.517,Z 249.912,A -85,B 0,C 180,E1 -5816.061,E2 -5816.061} C_VEL
LIN {X 0,Y 503.255,Z 256.495,A -85,B 0,C 180,E1 -5818.889,E2 -5818.889} C_VEL
LIN {X 0,Y 503.032,Z 263.163,A -85,B 0,C 180,E1 -5821.666,E2 -5821.666} C_VEL
LIN {X 0,Y 502.816,Z 270.837,A -85,B 0,C 180,E1 -5824.767,E2 -5824.767} C_VEL
LIN {X 0,Y 502.636,Z 278.578,A -85,B 0,C 180,E1 -5827.82,E2 -5827.82} C_VEL
LIN {X 0,Y 502.517,Z 286.378,A -85,B 0,C 180,E1 -5830.813,E2 -5830.813} C_VEL
LIN {X 0,Y 502.39,Z 295.317,A -85,B 0,C 180,E1 -5834.17,E2 -5834.17} C_VEL
LIN {X 0,Y 502.304,Z 299.424,A -85,B 0,C 180,E1 -5835.698,E2 -5835.698} C_VEL
LIN {X 0,Y 504.586,Z 314.05,A -85,B 0,C 180,E1 -5836.15,E2 -5836.15} C_VEL
LIN {X 0,Y 504.279,Z 326.993,A -85,B 0,C 180,E1 -5836.654,E2 -5836.654} C_VEL
LIN {X 0,Y 503.926,Z 338.902,A -85,B 0,C 180,E1 -5837.284,E2 -5837.284} C_VEL
LIN {X 0,Y 503.541,Z 349.664,A -85,B 0,C 180,E1 -5838.018,E2 -5838.018} C_VEL
LIN {X 0,Y 503.27,Z 360.363,A -85,B 0,C 180,E1 -5838.93,E2 -5838.93} C_VEL
LIN {X 0,Y 502.874,Z 370.001,A -85,B 0,C 180,E1 -5839.939,E2 -5839.939} C_VEL
LIN {X 0,Y 502.66,Z 377.909,A -85,B 0,C 180,E1 -5840.95,E2 -5840.95} C_VEL
LIN {X 0,Y 502.41,Z 385.632,A -85,B 0,C 180,E1 -5842.161,E2 -5842.161} C_VEL
LIN {X 0,Y 502.238,Z 392.335,A -85,B 0,C 180,E1 -5843.482,E2 -5843.482} C_VEL
LIN {X 0,Y 502.175,Z 397.477,A -85,B 0,C 180,E1 -5844.781,E2 -5844.781} C_VEL
LIN {X 0,Y 502.139,Z 401.093,A -85,B 0,C 180,E1 -5845.987,E2 -5845.987} C_VEL
LIN {X 0,Y 502.121,Z 402.958,A -85,B 0,C 180,E1 -5846.79,E2 -5846.79} C_VEL
LIN {X 0,Y 502.092,Z 404.355,A -85,B 0,C 180,E1 -5847.593,E2 -5847.593} C_VEL
LIN {X 0,Y 501.991,Z 405.955,A -85,B 0,C 180,E1 -5849.198,E2 -5849.198} C_VEL
LIN {X 0,Y 501.98,Z 406.169,A -85,B 0,C 180,E1 -5850,E2 -5850} C_VEL
LIN {X 0,Y 502.037,Z 405.34,A -85,B 0,C 180,E1 -5851.604,E2 -5851.604} C_VEL
LIN {X 0,Y 502.092,Z 404.34,A -85,B 0,C 180,E1 -5852.407,E2 -5852.407} C_VEL
LIN {X 0,Y 502.121,Z 402.936,A -85,B 0,C 180,E1 -5853.209,E2 -5853.209} C_VEL
LIN {X 0,Y 502.103,Z 399.986,A -85,B 0,C 180,E1 -5854.415,E2 -5854.415} C_VEL
LIN {X 0,Y 502.212,Z 395.996,A -85,B 0,C 180,E1 -5855.621,E2 -5855.621} C_VEL
LIN {X 0,Y 502.334,Z 389.959,A -85,B 0,C 180,E1 -5857.011,E2 -5857.011} C_VEL
LIN {X 0,Y 502.483,Z 383.149,A -85,B 0,C 180,E1 -5858.242,E2 -5858.242} C_VEL
LIN {X 0,Y 502.736,Z 374.827,A -85,B 0,C 180,E1 -5859.454,E2 -5859.454} C_VEL
LIN {X 0,Y 503.002,Z 366.291,A -85,B 0,C 180,E1 -5860.465,E2 -5860.465} C_VEL
LIN {X 0,Y 503.381,Z 355.751,A -85,B 0,C 180,E1 -5861.475,E2 -5861.475} C_VEL
LIN {X 0,Y 503.663,Z 344.828,A -85,B 0,C 180,E1 -5862.322,E2 -5862.322} C_VEL
LIN {X 0,Y 504.052,Z 333.907,A -85,B 0,C 180,E1 -5862.993,E2 -5862.993} C_VEL
LIN {X 0,Y 504.395,Z 322.157,A -85,B 0,C 180,E1 -5863.547,E2 -5863.547} C_VEL
LIN {X 0,Y 504.343,Z 312.281,A -85,B 0,C 180,E1 -5863.908,E2 -5863.908} C_VEL
LIN {X 0,Y 502.292,Z 299.198,A -85,B 0,C 180,E1 -5864.302,E2 -5864.302} C_VEL
LIN {X 0,Y 502.407,Z 290.566,A -85,B 0,C 180,E1 -5867.503,E2 -5867.503} C_VEL
LIN {X 0,Y 502.546,Z 282.736,A -85,B 0,C 180,E1 -5870.464,E2 -5870.464} C_VEL
LIN {X 0,Y 502.659,Z 274.922,A -85,B 0,C 180,E1 -5873.482,E2 -5873.482} C_VEL
LIN {X 0,Y 502.844,Z 268.301,A -85,B 0,C 180,E1 -5876.117,E2 -5876.117} C_VEL
LIN {X 0,Y 503.116,Z 260.638,A -85,B 0,C 180,E1 -5879.268,E2 -5879.268} C_VEL
LIN {X 0,Y 503.35,Z 253.088,A -85,B 0,C 180,E1 -5882.516,E2 -5882.516} C_VEL
LIN {X 0,Y 503.586,Z 246.725,A -85,B 0,C 180,E1 -5885.391,E2 -5885.391} C_VEL
LIN {X 0,Y 503.185,Z 242.946,A -85,B 0,C 180,E1 -5887.238,E2 -5887.238} C_VEL
LIN {X 0,Y 502.814,Z 240.856,A -85,B 0,C 180,E1 -5888.364,E2 -5888.364} C_VEL
LIN {X 0,Y 502.819,Z 240.855,A -85,B 0,C 180,E1 -5891.065,E2 -5891.065} C_VEL
LIN {X 0,Y 502.781,Z 240.861,A -85,B 0,C 180,E1 -5893.375,E2 -5893.375} C_VEL
LIN {X 0,Y 502.789,Z 240.859,A -85,B 0,C 180,E1 -5895.66,E2 -5895.66} C_VEL
LIN {X 0,Y 502.825,Z 240.854,A -85,B 0,C 180,E1 -5899.003,E2 -5899.003} C_VEL
LIN {X 0,Y 502.794,Z 240.857,A -85,B 0,C 180,E1 -5902.045,E2 -5902.045} C_VEL
LIN {X 0,Y 502.807,Z 240.855,A -85,B 0,C 180,E1 -5905.034,E2 -5905.034} C_VEL
LIN {X 0,Y 502.784,Z 240.859,A -85,B 0,C 180,E1 -5907.915,E2 -5907.915} C_VEL
LIN {X 0,Y 502.835,Z 240.853,A -85,B 0,C 180,E1 -5910.712,E2 -5910.712} C_VEL
LIN {X 0,Y 502.858,Z 240.848,A -85,B 0,C 180,E1 -5913.438,E2 -5913.438} C_VEL
LIN {X 0,Y 502.786,Z 240.859,A -85,B 0,C 180,E1 -5916.085,E2 -5916.085} C_VEL
LIN {X 0,Y 502.778,Z 240.859,A -85,B 0,C 180,E1 -5918.688,E2 -5918.688} C_VEL
LIN {X 0,Y 502.825,Z 240.854,A -85,B 0,C 180,E1 -5921.247,E2 -5921.247} C_VEL
LIN {X 0,Y 502.817,Z 240.854,A -85,B 0,C 180,E1 -5923.766,E2 -5923.766} C_VEL
LIN {X 0,Y 502.825,Z 240.854,A -85,B 0,C 180,E1 -5926.254,E2 -5926.254} C_VEL
LIN {X 0,Y 502.875,Z 240.846,A -85,B 0,C 180,E1 -5928.716,E2 -5928.716} C_VEL
LIN {X 0,Y 502.895,Z 240.844,A -85,B 0,C 180,E1 -5931.966,E2 -5931.966} C_VEL
LIN {X 0,Y 502.932,Z 240.841,A -85,B 0,C 180,E1 -5934.386,E2 -5934.386} C_VEL
LIN {X 0,Y 503.017,Z 240.831,A -85,B 0,C 180,E1 -5937.597,E2 -5937.597} C_VEL
LIN {X 0,Y 503.018,Z 240.829,A -85,B 0,C 180,E1 -5939.999,E2 -5939.999} C_VEL
LIN {X 0,Y 503.018,Z 240.83,A -85,B 0,C 180,E1 -5942.401,E2 -5942.401} C_VEL
LIN {X 0,Y 502.931,Z 240.841,A -85,B 0,C 180,E1 -5945.613,E2 -5945.613} C_VEL
LIN {X 0,Y 502.892,Z 240.846,A -85,B 0,C 180,E1 -5948.032,E2 -5948.032} C_VEL
LIN {X 0,Y 502.737,Z 240.89,A -85,B 0,C 180,E1 -5950.47,E2 -5950.47} C_VEL
LIN {X 0,Y 502.762,Z 244.424,A -85,B 0,C 180,E1 -5952.923,E2 -5952.923} C_VEL
LIN {X 0,Y 502.683,Z 248.093,A -85,B 0,C 180,E1 -5955.404,E2 -5955.404} C_VEL
LIN {X 0,Y 502.578,Z 252.062,A -85,B 0,C 180,E1 -5958.032,E2 -5958.032} C_VEL
LIN {X 0,Y 502.446,Z 257.131,A -85,B 0,C 180,E1 -5961.325,E2 -5961.325} C_VEL
LIN {X 0,Y 502.344,Z 261.23,A -85,B 0,C 180,E1 -5963.935,E2 -5963.935} C_VEL
LIN {X 0,Y 502.293,Z 265.483,A -85,B 0,C 180,E1 -5966.597,E2 -5966.597} C_VEL
LIN {X 0,Y 502.184,Z 269.912,A -85,B 0,C 180,E1 -5969.327,E2 -5969.327} C_VEL
LIN {X 0,Y 502.195,Z 274.071,A -85,B 0,C 180,E1 -5971.794,E2 -5971.794} C_VEL
LIN {X 0,Y 504.573,Z 286.303,A -85,B 0,C 180,E1 -5972.191,E2 -5972.191} C_VEL
LIN {X 0,Y 504.382,Z 298.775,A -85,B 0,C 180,E1 -5972.678,E2 -5972.678} C_VEL
LIN {X 0,Y 504.039,Z 311.083,A -85,B 0,C 180,E1 -5973.326,E2 -5973.326} C_VEL
LIN {X 0,Y 503.669,Z 322.892,A -85,B 0,C 180,E1 -5974.144,E2 -5974.144} C_VEL
LIN {X 0,Y 503.343,Z 333.229,A -85,B 0,C 180,E1 -5975.043,E2 -5975.043} C_VEL
LIN {X 0,Y 503.009,Z 342.686,A -85,B 0,C 180,E1 -5976.054,E2 -5976.054} C_VEL
LIN {X 0,Y 502.732,Z 351.148,A -85,B 0,C 180,E1 -5977.172,E2 -5977.172} C_VEL
LIN {X 0,Y 502.483,Z 358.901,A -85,B 0,C 180,E1 -5978.443,E2 -5978.443} C_VEL
LIN {X 0,Y 502.307,Z 364.963,A -85,B 0,C 180,E1 -5979.69,E2 -5979.69} C_VEL
LIN {X 0,Y 502.193,Z 370.313,A -85,B 0,C 180,E1 -5981.127,E2 -5981.127} C_VEL
LIN {X 0,Y 502.089,Z 373.365,A -85,B 0,C 180,E1 -5982.211,E2 -5982.211} C_VEL
LIN {X 0,Y 501.999,Z 375.608,A -85,B 0,C 180,E1 -5983.313,E2 -5983.313} C_VEL
LIN {X 0,Y 502.025,Z 377.106,A -85,B 0,C 180,E1 -5984.443,E2 -5984.443} C_VEL
LIN {X 0,Y 501.998,Z 377.828,A -85,B 0,C 180,E1 -5985.574,E2 -5985.574} C_VEL
LIN {X 0,Y 501.972,Z 377.678,A -85,B 0,C 180,E1 -5986.839,E2 -5986.839} C_VEL
LIN {X 0,Y 501.99,Z 376.838,A -85,B 0,C 180,E1 -5987.901,E2 -5987.901} C_VEL
LIN {X 0,Y 502.049,Z 374.991,A -85,B 0,C 180,E1 -5989.104,E2 -5989.104} C_VEL
LIN {X 0,Y 502.107,Z 372.281,A -85,B 0,C 180,E1 -5990.279,E2 -5990.279} C_VEL
LIN {X 0,Y 501.484,Z 370.49,A -85,B 0,C 180,E1 -5990.919,E2 -5990.919} C_VEL
LIN {X 0,Y 498.715,Z 367.13,A -85,B 0,C 180,E1 -5991.941,E2 -5991.941} C_VEL
LIN {X 0,Y 495.965,Z 363.071,A -85,B 0,C 180,E1 -5992.938,E2 -5992.938} C_VEL
LIN {X 0,Y 495.379,Z 360.184,A -85,B 0,C 180,E1 -5993.533,E2 -5993.533} C_VEL
LIN {X 0,Y 495.575,Z 353.66,A -85,B 0,C 180,E1 -5994.679,E2 -5994.679} C_VEL
LIN {X 0,Y 495.923,Z 344.508,A -85,B 0,C 180,E1 -5995.961,E2 -5995.961} C_VEL
LIN {X 0,Y 496.292,Z 334.54,A -85,B 0,C 180,E1 -5997.083,E2 -5997.083} C_VEL
LIN {X 0,Y 496.603,Z 324.394,A -85,B 0,C 180,E1 -5998,E2 -5998} C_VEL
LIN {X 0,Y 496.945,Z 313.316,A -85,B 0,C 180,E1 -5998.805,E2 -5998.805} C_VEL
LIN {X 0,Y 497.357,Z 301.447,A -85,B 0,C 180,E1 -5999.479,E2 -5999.479} C_VEL
LIN {X 0,Y 497.741,Z 288.455,A -85,B 0,C 180,E1 -6000.019,E2 -6000.019} C_VEL
LIN {X 0,Y 495.769,Z 277.626,A -85,B 0,C 180,E1 -6000.401,E2 -6000.401} C_VEL
LIN {X 0,Y 495.026,Z 273.868,A -85,B 0,C 180,E1 -6000.527,E2 -6000.527} C_VEL
LIN {X 0,Y 495.123,Z 269.151,A -85,B 0,C 180,E1 -6003.409,E2 -6003.409} C_VEL
LIN {X 0,Y 495.199,Z 264.015,A -85,B 0,C 180,E1 -6006.586,E2 -6006.586} C_VEL
LIN {X 0,Y 495.325,Z 259.443,A -85,B 0,C 180,E1 -6009.46,E2 -6009.46} C_VEL
LIN {X 0,Y 495.399,Z 254.426,A -85,B 0,C 180,E1 -6012.668,E2 -6012.668} C_VEL
LIN {X 0,Y 495.498,Z 250.51,A -85,B 0,C 180,E1 -6015.209,E2 -6015.209} C_VEL
LIN {X 0,Y 495.674,Z 245.465,A -85,B 0,C 180,E1 -6018.551,E2 -6018.551} C_VEL
LIN {X 0,Y 495.666,Z 241.813,A -85,B 0,C 180,E1 -6021.027,E2 -6021.027} C_VEL
LIN {X 0,Y 495.864,Z 241.72,A -85,B 0,C 180,E1 -6023.49,E2 -6023.49} C_VEL
LIN {X 0,Y 495.835,Z 241.723,A -85,B 0,C 180,E1 -6026.75,E2 -6026.75} C_VEL
LIN {X 0,Y 495.997,Z 241.703,A -85,B 0,C 180,E1 -6029.188,E2 -6029.188} C_VEL
LIN {X 0,Y 495.861,Z 241.718,A -85,B 0,C 180,E1 -6031.624,E2 -6031.624} C_VEL
LIN {X 0,Y 495.836,Z 241.723,A -85,B 0,C 180,E1 -6033.25,E2 -6033.25} C_VEL
LIN {X 0,Y 495.869,Z 241.72,A -85,B 0,C 180,E1 -6036.51,E2 -6036.51} C_VEL
LIN {X 0,Y 495.836,Z 241.724,A -85,B 0,C 180,E1 -6038.97,E2 -6038.97} C_VEL
LIN {X 0,Y 495.841,Z 241.723,A -85,B 0,C 180,E1 -6042.275,E2 -6042.275} C_VEL
LIN {X 0,Y 495.797,Z 241.728,A -85,B 0,C 180,E1 -6045.624,E2 -6045.624} C_VEL
LIN {X 0,Y 495.795,Z 241.728,A -85,B 0,C 180,E1 -6048.248,E2 -6048.248} C_VEL
LIN {X 0,Y 495.765,Z 241.731,A -85,B 0,C 180,E1 -6050.756,E2 -6050.756} C_VEL
LIN {X 0,Y 495.75,Z 241.733,A -85,B 0,C 180,E1 -6053.387,E2 -6053.387} C_VEL
LIN {X 0,Y 495.789,Z 241.73,A -85,B 0,C 180,E1 -6056.068,E2 -6056.068} C_VEL
LIN {X 0,Y 495.769,Z 241.73,A -85,B 0,C 180,E1 -6058.814,E2 -6058.814} C_VEL
LIN {X 0,Y 495.748,Z 241.735,A -85,B 0,C 180,E1 -6061.726,E2 -6061.726} C_VEL
LIN {X 0,Y 495.765,Z 241.732,A -85,B 0,C 180,E1 -6064.696,E2 -6064.696} C_VEL
LIN {X 0,Y 495.722,Z 241.737,A -85,B 0,C 180,E1 -6067.562,E2 -6067.562} C_VEL
LIN {X 0,Y 495.782,Z 241.73,A -85,B 0,C 180,E1 -6070.052,E2 -6070.052} C_VEL
LIN {X 0,Y 495.753,Z 241.734,A -85,B 0,C 180,E1 -6072.879,E2 -6072.879} C_VEL
LIN {X 0,Y 495.726,Z 241.737,A -85,B 0,C 180,E1 -6076,E2 -6076} C_VEL
LIN {X 0,Y 495.757,Z 241.733,A -85,B 0,C 180,E1 -6078.706,E2 -6078.706} C_VEL
LIN {X 0,Y 495.753,Z 241.734,A -85,B 0,C 180,E1 -6081.41,E2 -6081.41} C_VEL
LIN {X 0,Y 495.747,Z 241.733,A -85,B 0,C 180,E1 -6084.464,E2 -6084.464} C_VEL
LIN {X 0,Y 495.759,Z 241.733,A -85,B 0,C 180,E1 -6087.406,E2 -6087.406} C_VEL
LIN {X 0,Y 495.771,Z 241.73,A -85,B 0,C 180,E1 -6090.255,E2 -6090.255} C_VEL
LIN {X 0,Y 495.824,Z 241.726,A -85,B 0,C 180,E1 -6093.249,E2 -6093.249} C_VEL
LIN {X 0,Y 495.742,Z 241.735,A -85,B 0,C 180,E1 -6095.726,E2 -6095.726} C_VEL
LIN {X 0,Y 495.735,Z 241.736,A -85,B 0,C 180,E1 -6098.372,E2 -6098.372} C_VEL
LIN {X 0,Y 495.776,Z 241.73,A -85,B 0,C 180,E1 -6100.972,E2 -6100.972} C_VEL
LIN {X 0,Y 495.772,Z 241.73,A -85,B 0,C 180,E1 -6103.531,E2 -6103.531} C_VEL
LIN {X 0,Y 495.784,Z 241.729,A -85,B 0,C 180,E1 -6106.057,E2 -6106.057} C_VEL
LIN {X 0,Y 495.847,Z 241.723,A -85,B 0,C 180,E1 -6108.556,E2 -6108.556} C_VEL
LIN {X 0,Y 495.866,Z 241.718,A -85,B 0,C 180,E1 -6111.853,E2 -6111.853} C_VEL
LIN {X 0,Y 495.888,Z 241.717,A -85,B 0,C 180,E1 -6114.307,E2 -6114.307} C_VEL
LIN {X 0,Y 495.987,Z 241.704,A -85,B 0,C 180,E1 -6117.565,E2 -6117.565} C_VEL
LIN {X 0,Y 495.99,Z 241.704,A -85,B 0,C 180,E1 -6120.001,E2 -6120.001} C_VEL
LIN {X 0,Y 495.988,Z 241.704,A -85,B 0,C 180,E1 -6122.437,E2 -6122.437} C_VEL
LIN {X 0,Y 495.89,Z 241.718,A -85,B 0,C 180,E1 -6125.694,E2 -6125.694} C_VEL
LIN {X 0,Y 495.867,Z 241.72,A -85,B 0,C 180,E1 -6128.149,E2 -6128.149} C_VEL
LIN {X 0,Y 495.863,Z 241.719,A -85,B 0,C 180,E1 -6131.446,E2 -6131.446} C_VEL
LIN {X 0,Y 495.785,Z 241.728,A -85,B 0,C 180,E1 -6134.784,E2 -6134.784} C_VEL
LIN {X 0,Y 495.782,Z 241.729,A -85,B 0,C 180,E1 -6137.32,E2 -6137.32} C_VEL
LIN {X 0,Y 495.768,Z 241.733,A -85,B 0,C 180,E1 -6139.891,E2 -6139.891} C_VEL
LIN {X 0,Y 495.758,Z 241.732,A -85,B 0,C 180,E1 -6142.862,E2 -6142.862} C_VEL
LIN {X 0,Y 495.788,Z 241.73,A -85,B 0,C 180,E1 -6146.069,E2 -6146.069} C_VEL
LIN {X 0,Y 495.769,Z 241.731,A -85,B 0,C 180,E1 -6148.816,E2 -6148.816} C_VEL
LIN {X 0,Y 495.752,Z 241.734,A -85,B 0,C 180,E1 -6151.726,E2 -6151.726} C_VEL
LIN {X 0,Y 495.767,Z 241.733,A -85,B 0,C 180,E1 -6154.695,E2 -6154.695} C_VEL
LIN {X 0,Y 495.73,Z 241.736,A -85,B 0,C 180,E1 -6157.562,E2 -6157.562} C_VEL
LIN {X 0,Y 495.766,Z 241.733,A -85,B 0,C 180,E1 -6160.701,E2 -6160.701} C_VEL
LIN {X 0,Y 495.727,Z 241.737,A -85,B 0,C 180,E1 -6164.003,E2 -6164.003} C_VEL
LIN {X 0,Y 495.726,Z 241.737,A -85,B 0,C 180,E1 -6167.118,E2 -6167.118} C_VEL
LIN {X 0,Y 495.76,Z 241.733,A -85,B 0,C 180,E1 -6169.954,E2 -6169.954} C_VEL
LIN {X 0,Y 495.801,Z 241.895,A -85,B 0,C 180,E1 -6171.802,E2 -6171.802} C_VEL
LIN {X 0,Y 496.449,Z 246.061,A -85,B 0,C 180,E1 -6173.797,E2 -6173.797} C_VEL
LIN {X 0,Y 496.503,Z 250.924,A -85,B 0,C 180,E1 -6176.005,E2 -6176.005} C_VEL
LIN {X 0,Y 496.237,Z 257.505,A -85,B 0,C 180,E1 -6178.874,E2 -6178.874} C_VEL
LIN {X 0,Y 496.029,Z 263.599,A -85,B 0,C 180,E1 -6181.457,E2 -6181.457} C_VEL
LIN {X 0,Y 495.766,Z 271.824,A -85,B 0,C 180,E1 -6184.832,E2 -6184.832} C_VEL
LIN {X 0,Y 495.59,Z 279.568,A -85,B 0,C 180,E1 -6187.927,E2 -6187.927} C_VEL
LIN {X 0,Y 495.439,Z 287.327,A -85,B 0,C 180,E1 -6190.958,E2 -6190.958} C_VEL
LIN {X 0,Y 495.305,Z 296.241,A -85,B 0,C 180,E1 -6194.36,E2 -6194.36} C_VEL
LIN {X 0,Y 495.238,Z 299.233,A -85,B 0,C 180,E1 -6195.489,E2 -6195.489} C_VEL
LIN {X 0,Y 497.606,Z 314.557,A -85,B 0,C 180,E1 -6195.977,E2 -6195.977} C_VEL
LIN {X 0,Y 497.346,Z 327.878,A -85,B 0,C 180,E1 -6196.517,E2 -6196.517} C_VEL
LIN {X 0,Y 496.975,Z 338.953,A -85,B 0,C 180,E1 -6197.121,E2 -6197.121} C_VEL
LIN {X 0,Y 496.517,Z 350.731,A -85,B 0,C 180,E1 -6197.949,E2 -6197.949} C_VEL
LIN {X 0,Y 496.242,Z 361.213,A -85,B 0,C 180,E1 -6198.874,E2 -6198.874} C_VEL
LIN {X 0,Y 495.853,Z 369.783,A -85,B 0,C 180,E1 -6199.795,E2 -6199.795} C_VEL
LIN {X 0,Y 495.62,Z 377.695,A -85,B 0,C 180,E1 -6200.821,E2 -6200.821} C_VEL
LIN {X 0,Y 495.359,Z 385.424,A -85,B 0,C 180,E1 -6202.049,E2 -6202.049} C_VEL
LIN {X 0,Y 495.166,Z 392.539,A -85,B 0,C 180,E1 -6203.48,E2 -6203.48} C_VEL
LIN {X 0,Y 495.107,Z 397.276,A -85,B 0,C 180,E1 -6204.706,E2 -6204.706} C_VEL
LIN {X 0,Y 495.032,Z 400.892,A -85,B 0,C 180,E1 -6205.929,E2 -6205.929} C_VEL
LIN {X 0,Y 495.042,Z 402.758,A -85,B 0,C 180,E1 -6206.745,E2 -6206.745} C_VEL
LIN {X 0,Y 494.999,Z 404.156,A -85,B 0,C 180,E1 -6207.559,E2 -6207.559} C_VEL
LIN {X 0,Y 494.963,Z 405.151,A -85,B 0,C 180,E1 -6208.373,E2 -6208.373} C_VEL
LIN {X 0,Y 494.898,Z 405.969,A -85,B 0,C 180,E1 -6210,E2 -6210} C_VEL
LIN {X 0,Y 494.963,Z 405.138,A -85,B 0,C 180,E1 -6211.627,E2 -6211.627} C_VEL
LIN {X 0,Y 494.999,Z 404.136,A -85,B 0,C 180,E1 -6212.441,E2 -6212.441} C_VEL
LIN {X 0,Y 495.042,Z 402.731,A -85,B 0,C 180,E1 -6213.255,E2 -6213.255} C_VEL
LIN {X 0,Y 495.008,Z 399.777,A -85,B 0,C 180,E1 -6214.478,E2 -6214.478} C_VEL
LIN {X 0,Y 495.129,Z 395.783,A -85,B 0,C 180,E1 -6215.702,E2 -6215.702} C_VEL
LIN {X 0,Y 495.258,Z 389.637,A -85,B 0,C 180,E1 -6217.132,E2 -6217.132} C_VEL
LIN {X 0,Y 495.43,Z 382.922,A -85,B 0,C 180,E1 -6218.36,E2 -6218.36} C_VEL
LIN {X 0,Y 495.706,Z 374.594,A -85,B 0,C 180,E1 -6219.589,E2 -6219.589} C_VEL
LIN {X 0,Y 495.999,Z 366.049,A -85,B 0,C 180,E1 -6220.614,E2 -6220.614} C_VEL
LIN {X 0,Y 496.402,Z 355.502,A -85,B 0,C 180,E1 -6221.639,E2 -6221.639} C_VEL
LIN {X 0,Y 496.727,Z 344.394,A -85,B 0,C 180,E1 -6222.509,E2 -6222.509} C_VEL
LIN {X 0,Y 497.113,Z 333.644,A -85,B 0,C 180,E1 -6223.177,E2 -6223.177} C_VEL
LIN {X 0,Y 497.501,Z 320.597,A -85,B 0,C 180,E1 -6223.791,E2 -6223.791} C_VEL
LIN {X 0,Y 497.411,Z 313.176,A -85,B 0,C 180,E1 -6224.067,E2 -6224.067} C_VEL
LIN {X 0,Y 495.299,Z 299.884,A -85,B 0,C 180,E1 -6224.476,E2 -6224.476} C_VEL
LIN {X 0,Y 495.201,Z 298.909,A -85,B 0,C 180,E1 -6224.538,E2 -6224.538} C_VEL
LIN {X 0,Y 495.335,Z 291.497,A -85,B 0,C 180,E1 -6227.334,E2 -6227.334} C_VEL
LIN {X 0,Y 495.471,Z 283.052,A -85,B 0,C 180,E1 -6230.58,E2 -6230.58} C_VEL
LIN {X 0,Y 495.617,Z 275.881,A -85,B 0,C 180,E1 -6233.393,E2 -6233.393} C_VEL
LIN {X 0,Y 495.787,Z 269.276,A -85,B 0,C 180,E1 -6236.067,E2 -6236.067} C_VEL
LIN {X 0,Y 496.086,Z 260.562,A -85,B 0,C 180,E1 -6239.724,E2 -6239.724} C_VEL
LIN {X 0,Y 496.348,Z 254.119,A -85,B 0,C 180,E1 -6242.551,E2 -6242.551} C_VEL
LIN {X 0,Y 496.597,Z 247.785,A -85,B 0,C 180,E1 -6245.467,E2 -6245.467} C_VEL
LIN {X 0,Y 496.117,Z 243.66,A -85,B 0,C 180,E1 -6247.526,E2 -6247.526} C_VEL
LIN {X 0,Y 495.755,Z 241.735,A -85,B 0,C 180,E1 -6248.59,E2 -6248.59} C_VEL
LIN {X 0,Y 495.777,Z 241.731,A -85,B 0,C 180,E1 -6251.778,E2 -6251.778} C_VEL
LIN {X 0,Y 495.748,Z 241.735,A -85,B 0,C 180,E1 -6255.138,E2 -6255.138} C_VEL
LIN {X 0,Y 495.758,Z 241.734,A -85,B 0,C 180,E1 -6258.218,E2 -6258.218} C_VEL
LIN {X 0,Y 495.767,Z 241.733,A -85,B 0,C 180,E1 -6261.23,E2 -6261.23} C_VEL
LIN {X 0,Y 495.755,Z 241.734,A -85,B 0,C 180,E1 -6264.462,E2 -6264.462} C_VEL
LIN {X 0,Y 495.766,Z 241.732,A -85,B 0,C 180,E1 -6267.405,E2 -6267.405} C_VEL
LIN {X 0,Y 495.778,Z 241.73,A -85,B 0,C 180,E1 -6270.254,E2 -6270.254} C_VEL
LIN {X 0,Y 495.819,Z 241.725,A -85,B 0,C 180,E1 -6273.25,E2 -6273.25} C_VEL
LIN {X 0,Y 495.747,Z 241.735,A -85,B 0,C 180,E1 -6275.724,E2 -6275.724} C_VEL
LIN {X 0,Y 495.737,Z 241.736,A -85,B 0,C 180,E1 -6278.37,E2 -6278.37} C_VEL
LIN {X 0,Y 495.779,Z 241.732,A -85,B 0,C 180,E1 -6280.971,E2 -6280.971} C_VEL
LIN {X 0,Y 495.775,Z 241.731,A -85,B 0,C 180,E1 -6283.529,E2 -6283.529} C_VEL
LIN {X 0,Y 495.788,Z 241.731,A -85,B 0,C 180,E1 -6286.055,E2 -6286.055} C_VEL
LIN {X 0,Y 495.848,Z 241.722,A -85,B 0,C 180,E1 -6288.554,E2 -6288.554} C_VEL
LIN {X 0,Y 495.867,Z 241.72,A -85,B 0,C 180,E1 -6291.851,E2 -6291.851} C_VEL
LIN {X 0,Y 495.89,Z 241.718,A -85,B 0,C 180,E1 -6294.306,E2 -6294.306} C_VEL
LIN {X 0,Y 495.986,Z 241.707,A -85,B 0,C 180,E1 -6297.563,E2 -6297.563} C_VEL
LIN {X 0,Y 495.989,Z 241.704,A -85,B 0,C 180,E1 -6299.999,E2 -6299.999} C_VEL
LIN {X 0,Y 495.986,Z 241.706,A -85,B 0,C 180,E1 -6302.435,E2 -6302.435} C_VEL
LIN {X 0,Y 495.889,Z 241.719,A -85,B 0,C 180,E1 -6305.693,E2 -6305.693} C_VEL
LIN {X 0,Y 495.863,Z 241.721,A -85,B 0,C 180,E1 -6308.147,E2 -6308.147} C_VEL
LIN {X 0,Y 495.761,Z 241.735,A -85,B 0,C 180,E1 -6309.793,E2 -6309.793} C_VEL
LIN {X 0,Y 495.71,Z 242.07,A -85,B 0,C 180,E1 -6310.62,E2 -6310.62} C_VEL
LIN {X 0,Y 495.711,Z 245.617,A -85,B 0,C 180,E1 -6313.11,E2 -6313.11} C_VEL
LIN {X 0,Y 495.631,Z 249.297,A -85,B 0,C 180,E1 -6315.628,E2 -6315.628} C_VEL
LIN {X 0,Y 495.507,Z 253.09,A -85,B 0,C 180,E1 -6318.181,E2 -6318.181} C_VEL
LIN {X 0,Y 495.398,Z 257.041,A -85,B 0,C 180,E1 -6320.772,E2 -6320.772} C_VEL
LIN {X 0,Y 495.289,Z 261.122,A -85,B 0,C 180,E1 -6323.409,E2 -6323.409} C_VEL
LIN {X 0,Y 495.254,Z 265.348,A -85,B 0,C 180,E1 -6326.097,E2 -6326.097} C_VEL
LIN {X 0,Y 495.122,Z 269.752,A -85,B 0,C 180,E1 -6328.855,E2 -6328.855} C_VEL
LIN {X 0,Y 495.096,Z 274.161,A -85,B 0,C 180,E1 -6331.574,E2 -6331.574} C_VEL
LIN {X 0,Y 497.717,Z 287.824,A -85,B 0,C 180,E1 -6332.043,E2 -6332.043} C_VEL
LIN {X 0,Y 497.457,Z 301.089,A -85,B 0,C 180,E1 -6332.589,E2 -6332.589} C_VEL
LIN {X 0,Y 497.103,Z 312.372,A -85,B 0,C 180,E1 -6333.218,E2 -6333.218} C_VEL
LIN {X 0,Y 496.741,Z 323.054,A -85,B 0,C 180,E1 -6333.975,E2 -6333.975} C_VEL
LIN {X 0,Y 496.355,Z 333.58,A -85,B 0,C 180,E1 -6334.903,E2 -6334.903} C_VEL
LIN {X 0,Y 495.981,Z 343.228,A -85,B 0,C 180,E1 -6335.955,E2 -6335.955} C_VEL
LIN {X 0,Y 495.641,Z 352.392,A -85,B 0,C 180,E1 -6337.205,E2 -6337.205} C_VEL
LIN {X 0,Y 495.426,Z 359.235,A -85,B 0,C 180,E1 -6338.36,E2 -6338.36} C_VEL
LIN {X 0,Y 495.225,Z 365.543,A -85,B 0,C 180,E1 -6339.687,E2 -6339.687} C_VEL
LIN {X 0,Y 495.118,Z 369.562,A -85,B 0,C 180,E1 -6340.763,E2 -6340.763} C_VEL
LIN {X 0,Y 495.046,Z 372.783,A -85,B 0,C 180,E1 -6341.853,E2 -6341.853} C_VEL
LIN {X 0,Y 494.948,Z 375.262,A -85,B 0,C 180,E1 -6342.965,E2 -6342.965} C_VEL
LIN {X 0,Y 494.914,Z 376.982,A -85,B 0,C 180,E1 -6344.091,E2 -6344.091} C_VEL
LIN {X 0,Y 494.916,Z 377.903,A -85,B 0,C 180,E1 -6345.235,E2 -6345.235} C_VEL
LIN {X 0,Y 494.881,Z 378.047,A -85,B 0,C 180,E1 -6346.406,E2 -6346.406} C_VEL
LIN {X 0,Y 494.89,Z 377.361,A -85,B 0,C 180,E1 -6347.598,E2 -6347.598} C_VEL
LIN {X 0,Y 494.958,Z 375.056,A -85,B 0,C 180,E1 -6349.221,E2 -6349.221} C_VEL
LIN {X 0,Y 495.04,Z 372.59,A -85,B 0,C 180,E1 -6350.294,E2 -6350.294} C_VEL
LIN {X 0,Y 495.175,Z 367.567,A -85,B 0,C 180,E1 -6351.875,E2 -6351.875} C_VEL
LIN {X 0,Y 495.294,Z 362.72,A -85,B 0,C 180,E1 -6353.024,E2 -6353.024} C_VEL
LIN {X 0,Y 495.379,Z 360.184,A -85,B 0,C 180,E1 -6353.533,E2 -6353.533} C_VEL
LIN {X 0,Y 494.805,Z 357.134,A -85,B 0,C 180,E1 -6354.114,E2 -6354.114} C_VEL
LIN {X 0,Y 492.138,Z 351.853,A -85,B 0,C 180,E1 -6355.042,E2 -6355.042} C_VEL
LIN {X 0,Y 489.529,Z 346.006,A -85,B 0,C 180,E1 -6355.927,E2 -6355.927} C_VEL
LIN {X 0,Y 489.043,Z 342.01,A -85,B 0,C 180,E1 -6356.433,E2 -6356.433} C_VEL
LIN {X 0,Y 489.452,Z 331.602,A -85,B 0,C 180,E1 -6357.545,E2 -6357.545} C_VEL
LIN {X 0,Y 489.769,Z 321.52,A -85,B 0,C 180,E1 -6358.416,E2 -6358.416} C_VEL
LIN {X 0,Y 490.173,Z 309.678,A -85,B 0,C 180,E1 -6359.224,E2 -6359.224} C_VEL
LIN {X 0,Y 490.603,Z 297.514,A -85,B 0,C 180,E1 -6359.861,E2 -6359.861} C_VEL
LIN {X 0,Y 490.708,Z 288.031,A -85,B 0,C 180,E1 -6360.242,E2 -6360.242} C_VEL
LIN {X 0,Y 487.973,Z 274.042,A -85,B 0,C 180,E1 -6360.735,E2 -6360.735} C_VEL
LIN {X 0,Y 488.059,Z 269.592,A -85,B 0,C 180,E1 -6363.488,E2 -6363.488} C_VEL
LIN {X 0,Y 488.167,Z 263.784,A -85,B 0,C 180,E1 -6367.126,E2 -6367.126} C_VEL
LIN {X 0,Y 488.285,Z 259.597,A -85,B 0,C 180,E1 -6369.792,E2 -6369.792} C_VEL
LIN {X 0,Y 488.33,Z 255.555,A -85,B 0,C 180,E1 -6372.409,E2 -6372.409} C_VEL
LIN {X 0,Y 488.425,Z 251.616,A -85,B 0,C 180,E1 -6374.989,E2 -6374.989} C_VEL
LIN {X 0,Y 488.611,Z 246.529,A -85,B 0,C 180,E1 -6378.383,E2 -6378.383} C_VEL
LIN {X 0,Y 488.626,Z 242.869,A -85,B 0,C 180,E1 -6380.897,E2 -6380.897} C_VEL
LIN {X 0,Y 488.822,Z 242.597,A -85,B 0,C 180,E1 -6382.755,E2 -6382.755} C_VEL
LIN {X 0,Y 488.802,Z 242.599,A -85,B 0,C 180,E1 -6385.051,E2 -6385.051} C_VEL
LIN {X 0,Y 488.95,Z 242.58,A -85,B 0,C 180,E1 -6387.529,E2 -6387.529} C_VEL
LIN {X 0,Y 488.958,Z 242.58,A -85,B 0,C 180,E1 -6390,E2 -6390} C_VEL
LIN {X 0,Y 488.953,Z 242.581,A -85,B 0,C 180,E1 -6392.471,E2 -6392.471} C_VEL
LIN {X 0,Y 488.846,Z 242.595,A -85,B 0,C 180,E1 -6395.776,E2 -6395.776} C_VEL
LIN {X 0,Y 488.808,Z 242.6,A -85,B 0,C 180,E1 -6398.266,E2 -6398.266} C_VEL
LIN {X 0,Y 488.82,Z 242.597,A -85,B 0,C 180,E1 -6401.612,E2 -6401.612} C_VEL
LIN {X 0,Y 488.751,Z 242.606,A -85,B 0,C 180,E1 -6405.001,E2 -6405.001} C_VEL
LIN {X 0,Y 488.744,Z 242.607,A -85,B 0,C 180,E1 -6408.442,E2 -6408.442} C_VEL
LIN {X 0,Y 488.73,Z 242.608,A -85,B 0,C 180,E1 -6411.069,E2 -6411.069} C_VEL
LIN {X 0,Y 488.691,Z 242.615,A -85,B 0,C 180,E1 -6413.745,E2 -6413.745} C_VEL
LIN {X 0,Y 488.788,Z 242.6,A -85,B 0,C 180,E1 -6416.946,E2 -6416.946} C_VEL
LIN {X 0,Y 488.708,Z 242.611,A -85,B 0,C 180,E1 -6420.365,E2 -6420.365} C_VEL
LIN {X 0,Y 488.724,Z 242.61,A -85,B 0,C 180,E1 -6423.485,E2 -6423.485} C_VEL
LIN {X 0,Y 488.677,Z 242.614,A -85,B 0,C 180,E1 -6426.356,E2 -6426.356} C_VEL
LIN {X 0,Y 488.737,Z 242.609,A -85,B 0,C 180,E1 -6429.25,E2 -6429.25} C_VEL
LIN {X 0,Y 488.724,Z 242.608,A -85,B 0,C 180,E1 -6432.521,E2 -6432.521} C_VEL
LIN {X 0,Y 488.691,Z 242.613,A -85,B 0,C 180,E1 -6435.976,E2 -6435.976} C_VEL
LIN {X 0,Y 488.712,Z 242.609,A -85,B 0,C 180,E1 -6438.587,E2 -6438.587} C_VEL
LIN {X 0,Y 488.736,Z 242.607,A -85,B 0,C 180,E1 -6440.942,E2 -6440.942} C_VEL
LIN {X 0,Y 488.675,Z 242.614,A -85,B 0,C 180,E1 -6443.869,E2 -6443.869} C_VEL
LIN {X 0,Y 488.728,Z 242.609,A -85,B 0,C 180,E1 -6446.878,E2 -6446.878} C_VEL
LIN {X 0,Y 488.724,Z 242.608,A -85,B 0,C 180,E1 -6449.782,E2 -6449.782} C_VEL
LIN {X 0,Y 488.789,Z 242.602,A -85,B 0,C 180,E1 -6453.055,E2 -6453.055} C_VEL
LIN {X 0,Y 488.684,Z 242.613,A -85,B 0,C 180,E1 -6456.255,E2 -6456.255} C_VEL
LIN {X 0,Y 488.736,Z 242.609,A -85,B 0,C 180,E1 -6459.176,E2 -6459.176} C_VEL
LIN {X 0,Y 488.75,Z 242.606,A -85,B 0,C 180,E1 -6461.629,E2 -6461.629} C_VEL
LIN {X 0,Y 488.753,Z 242.607,A -85,B 0,C 180,E1 -6465,E2 -6465} C_VEL
LIN {X 0,Y 488.8,Z 242.6,A -85,B 0,C 180,E1 -6468.389,E2 -6468.389} C_VEL
LIN {X 0,Y 488.811,Z 242.597,A -85,B 0,C 180,E1 -6471.735,E2 -6471.735} C_VEL
LIN {X 0,Y 488.847,Z 242.594,A -85,B 0,C 180,E1 -6474.225,E2 -6474.225} C_VEL
LIN {X 0,Y 488.954,Z 242.581,A -85,B 0,C 180,E1 -6477.53,E2 -6477.53} C_VEL
LIN {X 0,Y 488.949,Z 242.581,A -85,B 0,C 180,E1 -6480.825,E2 -6480.825} C_VEL
LIN {X 0,Y 488.956,Z 242.58,A -85,B 0,C 180,E1 -6482.472,E2 -6482.472} C_VEL
LIN {X 0,Y 488.849,Z 242.595,A -85,B 0,C 180,E1 -6485.777,E2 -6485.777} C_VEL
LIN {X 0,Y 488.811,Z 242.598,A -85,B 0,C 180,E1 -6488.267,E2 -6488.267} C_VEL
LIN {X 0,Y 488.824,Z 242.598,A -85,B 0,C 180,E1 -6491.613,E2 -6491.613} C_VEL
LIN {X 0,Y 488.757,Z 242.604,A -85,B 0,C 180,E1 -6495.001,E2 -6495.001} C_VEL
LIN {X 0,Y 488.751,Z 242.606,A -85,B 0,C 180,E1 -6498.443,E2 -6498.443} C_VEL
LIN {X 0,Y 488.703,Z 242.611,A -85,B 0,C 180,E1 -6501.072,E2 -6501.072} C_VEL
LIN {X 0,Y 488.689,Z 242.615,A -85,B 0,C 180,E1 -6503.746,E2 -6503.746} C_VEL
LIN {X 0,Y 488.789,Z 242.6,A -85,B 0,C 180,E1 -6506.945,E2 -6506.945} C_VEL
LIN {X 0,Y 488.707,Z 242.61,A -85,B 0,C 180,E1 -6510.364,E2 -6510.364} C_VEL
LIN {X 0,Y 488.728,Z 242.609,A -85,B 0,C 180,E1 -6513.484,E2 -6513.484} C_VEL
LIN {X 0,Y 488.686,Z 242.612,A -85,B 0,C 180,E1 -6516.356,E2 -6516.356} C_VEL
LIN {X 0,Y 488.7,Z 242.614,A -85,B 0,C 180,E1 -6519.255,E2 -6519.255} C_VEL
LIN {X 0,Y 488.706,Z 242.612,A -85,B 0,C 180,E1 -6521.601,E2 -6521.601} C_VEL
LIN {X 0,Y 488.701,Z 242.612,A -85,B 0,C 180,E1 -6524.804,E2 -6524.804} C_VEL
LIN {X 0,Y 488.692,Z 242.615,A -85,B 0,C 180,E1 -6527.475,E2 -6527.475} C_VEL
LIN {X 0,Y 488.734,Z 242.607,A -85,B 0,C 180,E1 -6529.677,E2 -6529.677} C_VEL
LIN {X 0,Y 488.737,Z 242.618,A -85,B 0,C 180,E1 -6531.543,E2 -6531.543} C_VEL
LIN {X 0,Y 489.486,Z 247.542,A -85,B 0,C 180,E1 -6533.938,E2 -6533.938} C_VEL
LIN {X 0,Y 489.481,Z 252.881,A -85,B 0,C 180,E1 -6536.385,E2 -6536.385} C_VEL
LIN {X 0,Y 489.16,Z 260.08,A -85,B 0,C 180,E1 -6539.548,E2 -6539.548} C_VEL
LIN {X 0,Y 488.888,Z 266.187,A -85,B 0,C 180,E1 -6542.148,E2 -6542.148} C_VEL
LIN {X 0,Y 488.72,Z 272.935,A -85,B 0,C 180,E1 -6544.955,E2 -6544.955} C_VEL
LIN {X 0,Y 488.512,Z 280.551,A -85,B 0,C 180,E1 -6548.035,E2 -6548.035} C_VEL
LIN {X 0,Y 488.345,Z 288.291,A -85,B 0,C 180,E1 -6551.107,E2 -6551.107} C_VEL
LIN {X 0,Y 488.257,Z 296.056,A -85,B 0,C 180,E1 -6554.128,E2 -6554.128} C_VEL
LIN {X 0,Y 488.159,Z 299.039,A -85,B 0,C 180,E1 -6555.274,E2 -6555.274} C_VEL
LIN {X 0,Y 490.587,Z 314.673,A -85,B 0,C 180,E1 -6555.786,E2 -6555.786} C_VEL
LIN {X 0,Y 490.425,Z 327.631,A -85,B 0,C 180,E1 -6556.323,E2 -6556.323} C_VEL
LIN {X 0,Y 490.012,Z 339.184,A -85,B 0,C 180,E1 -6556.966,E2 -6556.966} C_VEL
LIN {X 0,Y 489.543,Z 350.504,A -85,B 0,C 180,E1 -6557.775,E2 -6557.775} C_VEL
LIN {X 0,Y 489.239,Z 360.991,A -85,B 0,C 180,E1 -6558.713,E2 -6558.713} C_VEL
LIN {X 0,Y 488.844,Z 369.566,A -85,B 0,C 180,E1 -6559.647,E2 -6559.647} C_VEL
LIN {X 0,Y 488.556,Z 377.481,A -85,B 0,C 180,E1 -6560.687,E2 -6560.687} C_VEL
LIN {X 0,Y 488.291,Z 385.216,A -85,B 0,C 180,E1 -6561.933,E2 -6561.933} C_VEL
LIN {X 0,Y 488.102,Z 392.335,A -85,B 0,C 180,E1 -6563.385,E2 -6563.385} C_VEL
LIN {X 0,Y 488.02,Z 397.073,A -85,B 0,C 180,E1 -6564.629,E2 -6564.629} C_VEL
LIN {X 0,Y 487.928,Z 400.691,A -85,B 0,C 180,E1 -6565.87,E2 -6565.87} C_VEL
LIN {X 0,Y 487.965,Z 402.559,A -85,B 0,C 180,E1 -6566.697,E2 -6566.697} C_VEL
LIN {X 0,Y 487.91,Z 403.957,A -85,B 0,C 180,E1 -6567.523,E2 -6567.523} C_VEL
LIN {X 0,Y 487.891,Z 404.952,A -85,B 0,C 180,E1 -6568.349,E2 -6568.349} C_VEL
LIN {X 0,Y 487.819,Z 405.77,A -85,B 0,C 180,E1 -6570,E2 -6570} C_VEL
LIN {X 0,Y 487.891,Z 404.936,A -85,B 0,C 180,E1 -6571.651,E2 -6571.651} C_VEL
LIN {X 0,Y 487.909,Z 403.932,A -85,B 0,C 180,E1 -6572.477,E2 -6572.477} C_VEL
LIN {X 0,Y 487.965,Z 402.526,A -85,B 0,C 180,E1 -6573.302,E2 -6573.302} C_VEL
LIN {X 0,Y 487.921,Z 399.568,A -85,B 0,C 180,E1 -6574.544,E2 -6574.544} C_VEL
LIN {X 0,Y 488.026,Z 395.568,A -85,B 0,C 180,E1 -6575.785,E2 -6575.785} C_VEL
LIN {X 0,Y 488.185,Z 389.415,A -85,B 0,C 180,E1 -6577.236,E2 -6577.236} C_VEL
LIN {X 0,Y 488.365,Z 382.694,A -85,B 0,C 180,E1 -6578.482,E2 -6578.482} C_VEL
LIN {X 0,Y 488.672,Z 374.363,A -85,B 0,C 180,E1 -6579.729,E2 -6579.729} C_VEL
LIN {X 0,Y 489.005,Z 365.813,A -85,B 0,C 180,E1 -6580.768,E2 -6580.768} C_VEL
LIN {X 0,Y 489.419,Z 355.261,A -85,B 0,C 180,E1 -6581.807,E2 -6581.807} C_VEL
LIN {X 0,Y 489.757,Z 343.829,A -85,B 0,C 180,E1 -6582.714,E2 -6582.714} C_VEL
LIN {X 0,Y 490.258,Z 331.444,A -85,B 0,C 180,E1 -6583.47,E2 -6583.47} C_VEL
LIN {X 0,Y 490.616,Z 319.062,A -85,B 0,C 180,E1 -6584.041,E2 -6584.041} C_VEL
LIN {X 0,Y 490.541,Z 314.445,A -85,B 0,C 180,E1 -6584.215,E2 -6584.215} C_VEL
LIN {X 0,Y 488.441,Z 300.809,A -85,B 0,C 180,E1 -6584.662,E2 -6584.662} C_VEL
LIN {X 0,Y 488.136,Z 298.777,A -85,B 0,C 180,E1 -6584.726,E2 -6584.726} C_VEL
LIN {X 0,Y 488.26,Z 291.311,A -85,B 0,C 180,E1 -6587.594,E2 -6587.594} C_VEL
LIN {X 0,Y 488.403,Z 283.334,A -85,B 0,C 180,E1 -6590.717,E2 -6590.717} C_VEL
LIN {X 0,Y 488.578,Z 275.769,A -85,B 0,C 180,E1 -6593.751,E2 -6593.751} C_VEL
LIN {X 0,Y 488.761,Z 269.156,A -85,B 0,C 180,E1 -6596.471,E2 -6596.471} C_VEL
LIN {X 0,Y 489.073,Z 261.574,A -85,B 0,C 180,E1 -6599.72,E2 -6599.72} C_VEL
LIN {X 0,Y 489.343,Z 255.146,A -85,B 0,C 180,E1 -6602.586,E2 -6602.586} C_VEL
LIN {X 0,Y 489.568,Z 249.791,A -85,B 0,C 180,E1 -6605.088,E2 -6605.088} C_VEL
LIN {X 0,Y 489.28,Z 245.745,A -85,B 0,C 180,E1 -6607.105,E2 -6607.105} C_VEL
LIN {X 0,Y 488.73,Z 242.611,A -85,B 0,C 180,E1 -6608.803,E2 -6608.803} C_VEL
LIN {X 0,Y 488.723,Z 242.611,A -85,B 0,C 180,E1 -6611.601,E2 -6611.601} C_VEL
LIN {X 0,Y 488.711,Z 242.611,A -85,B 0,C 180,E1 -6614.8,E2 -6614.8} C_VEL
LIN {X 0,Y 488.69,Z 242.617,A -85,B 0,C 180,E1 -6617.473,E2 -6617.473} C_VEL
LIN {X 0,Y 488.731,Z 242.611,A -85,B 0,C 180,E1 -6619.676,E2 -6619.676} C_VEL
LIN {X 0,Y 488.68,Z 242.616,A -85,B 0,C 180,E1 -6622.276,E2 -6622.276} C_VEL
LIN {X 0,Y 488.726,Z 242.609,A -85,B 0,C 180,E1 -6625.05,E2 -6625.05} C_VEL
LIN {X 0,Y 488.703,Z 242.612,A -85,B 0,C 180,E1 -6628.044,E2 -6628.044} C_VEL
LIN {X 0,Y 488.73,Z 242.61,A -85,B 0,C 180,E1 -6630.729,E2 -6630.729} C_VEL
LIN {X 0,Y 488.752,Z 242.605,A -85,B 0,C 180,E1 -6633.527,E2 -6633.527} C_VEL
LIN {X 0,Y 488.688,Z 242.614,A -85,B 0,C 180,E1 -6636.253,E2 -6636.253} C_VEL
LIN {X 0,Y 488.74,Z 242.609,A -85,B 0,C 180,E1 -6639.175,E2 -6639.175} C_VEL
LIN {X 0,Y 488.729,Z 242.609,A -85,B 0,C 180,E1 -6642.422,E2 -6642.422} C_VEL
LIN {X 0,Y 488.755,Z 242.606,A -85,B 0,C 180,E1 -6644.999,E2 -6644.999} C_VEL
LIN {X 0,Y 488.801,Z 242.601,A -85,B 0,C 180,E1 -6648.387,E2 -6648.387} C_VEL
LIN {X 0,Y 488.812,Z 242.599,A -85,B 0,C 180,E1 -6651.733,E2 -6651.733} C_VEL
LIN {X 0,Y 488.849,Z 242.595,A -85,B 0,C 180,E1 -6654.223,E2 -6654.223} C_VEL
LIN {X 0,Y 488.953,Z 242.583,A -85,B 0,C 180,E1 -6657.528,E2 -6657.528} C_VEL
LIN {X 0,Y 488.946,Z 242.582,A -85,B 0,C 180,E1 -6660.823,E2 -6660.823} C_VEL
LIN {X 0,Y 488.954,Z 242.582,A -85,B 0,C 180,E1 -6662.47,E2 -6662.47} C_VEL
LIN {X 0,Y 488.848,Z 242.596,A -85,B 0,C 180,E1 -6665.775,E2 -6665.775} C_VEL
LIN {X 0,Y 488.807,Z 242.6,A -85,B 0,C 180,E1 -6668.265,E2 -6668.265} C_VEL
LIN {X 0,Y 488.702,Z 242.615,A -85,B 0,C 180,E1 -6669.936,E2 -6669.936} C_VEL
LIN {X 0,Y 488.686,Z 243.266,A -85,B 0,C 180,E1 -6670.774,E2 -6670.774} C_VEL
LIN {X 0,Y 488.71,Z 245.608,A -85,B 0,C 180,E1 -6672.456,E2 -6672.456} C_VEL
LIN {X 0,Y 488.587,Z 249.957,A -85,B 0,C 180,E1 -6675.479,E2 -6675.479} C_VEL
LIN {X 0,Y 488.445,Z 254.336,A -85,B 0,C 180,E1 -6678.453,E2 -6678.453} C_VEL
LIN {X 0,Y 488.315,Z 258.269,A -85,B 0,C 180,E1 -6681.087,E2 -6681.087} C_VEL
LIN {X 0,Y 488.239,Z 262.398,A -85,B 0,C 180,E1 -6683.768,E2 -6683.768} C_VEL
LIN {X 0,Y 488.171,Z 267.111,A -85,B 0,C 180,E1 -6686.802,E2 -6686.802} C_VEL
LIN {X 0,Y 488.028,Z 271.098,A -85,B 0,C 180,E1 -6689.315,E2 -6689.315} C_VEL
LIN {X 0,Y 488.032,Z 274.371,A -85,B 0,C 180,E1 -6691.364,E2 -6691.364} C_VEL
LIN {X 0,Y 490.783,Z 288.197,A -85,B 0,C 180,E1 -6691.848,E2 -6691.848} C_VEL
LIN {X 0,Y 490.554,Z 301.034,A -85,B 0,C 180,E1 -6692.384,E2 -6692.384} C_VEL
LIN {X 0,Y 490.177,Z 312.232,A -85,B 0,C 180,E1 -6693.012,E2 -6693.012} C_VEL
LIN {X 0,Y 489.782,Z 323.479,A -85,B 0,C 180,E1 -6693.821,E2 -6693.821} C_VEL
LIN {X 0,Y 489.375,Z 334.304,A -85,B 0,C 180,E1 -6694.795,E2 -6694.795} C_VEL
LIN {X 0,Y 488.958,Z 343.76,A -85,B 0,C 180,E1 -6695.852,E2 -6695.852} C_VEL
LIN {X 0,Y 488.653,Z 351.758,A -85,B 0,C 180,E1 -6696.95,E2 -6696.95} C_VEL
LIN {X 0,Y 488.393,Z 359.301,A -85,B 0,C 180,E1 -6698.225,E2 -6698.225} C_VEL
LIN {X 0,Y 488.162,Z 365.503,A -85,B 0,C 180,E1 -6699.539,E2 -6699.539} C_VEL
LIN {X 0,Y 488.04,Z 370.564,A -85,B 0,C 180,E1 -6700.935,E2 -6700.935} C_VEL
LIN {X 0,Y 487.932,Z 373.636,A -85,B 0,C 180,E1 -6702.047,E2 -6702.047} C_VEL
LIN {X 0,Y 487.894,Z 375.109,A -85,B 0,C 180,E1 -6702.724,E2 -6702.724} C_VEL
LIN {X 0,Y 487.823,Z 376.997,A -85,B 0,C 180,E1 -6703.919,E2 -6703.919} C_VEL
LIN {X 0,Y 487.837,Z 378.032,A -85,B 0,C 180,E1 -6705.098,E2 -6705.098} C_VEL
LIN {X 0,Y 487.781,Z 378.279,A -85,B 0,C 180,E1 -6706.245,E2 -6706.245} C_VEL
LIN {X 0,Y 487.806,Z 377.786,A -85,B 0,C 180,E1 -6707.38,E2 -6707.38} C_VEL
LIN {X 0,Y 487.855,Z 376.506,A -85,B 0,C 180,E1 -6708.511,E2 -6708.511} C_VEL
LIN {X 0,Y 487.897,Z 374.204,A -85,B 0,C 180,E1 -6709.767,E2 -6709.767} C_VEL
LIN {X 0,Y 487.996,Z 370.828,A -85,B 0,C 180,E1 -6711.048,E2 -6711.048} C_VEL
LIN {X 0,Y 488.143,Z 366.208,A -85,B 0,C 180,E1 -6712.357,E2 -6712.357} C_VEL
LIN {X 0,Y 488.328,Z 360.096,A -85,B 0,C 180,E1 -6713.7,E2 -6713.7} C_VEL
LIN {X 0,Y 488.606,Z 352.106,A -85,B 0,C 180,E1 -6715.07,E2 -6715.07} C_VEL
LIN {X 0,Y 488.947,Z 343.83,A -85,B 0,C 180,E1 -6716.212,E2 -6716.212} C_VEL
LIN {X 0,Y 489.043,Z 342.01,A -85,B 0,C 180,E1 -6716.433,E2 -6716.433} C_VEL
LIN {X 0,Y 488.56,Z 337.89,A -85,B 0,C 180,E1 -6716.92,E2 -6716.92} C_VEL
LIN {X 0,Y 484.829,Z 328.098,A -85,B 0,C 180,E1 -6717.995,E2 -6717.995} C_VEL
LIN {X 0,Y 483.145,Z 322.015,A -85,B 0,C 180,E1 -6718.558,E2 -6718.558} C_VEL
LIN {X 0,Y 482.962,Z 318.698,A -85,B 0,C 180,E1 -6718.818,E2 -6718.818} C_VEL
LIN {X 0,Y 483.331,Z 306.924,A -85,B 0,C 180,E1 -6719.59,E2 -6719.59} C_VEL
LIN {X 0,Y 483.791,Z 295.366,A -85,B 0,C 180,E1 -6720.163,E2 -6720.163} C_VEL
LIN {X 0,Y 483.743,Z 288.726,A -85,B 0,C 180,E1 -6720.429,E2 -6720.429} C_VEL
LIN {X 0,Y 481.205,Z 275.973,A -85,B 0,C 180,E1 -6720.888,E2 -6720.888} C_VEL
LIN {X 0,Y 480.892,Z 274.224,A -85,B 0,C 180,E1 -6720.957,E2 -6720.957} C_VEL
LIN {X 0,Y 480.977,Z 269.358,A -85,B 0,C 180,E1 -6724.002,E2 -6724.002} C_VEL
LIN {X 0,Y 481.089,Z 264.665,A -85,B 0,C 180,E1 -6726.971,E2 -6726.971} C_VEL
LIN {X 0,Y 481.197,Z 260.765,A -85,B 0,C 180,E1 -6729.481,E2 -6729.481} C_VEL
LIN {X 0,Y 481.289,Z 256.673,A -85,B 0,C 180,E1 -6732.143,E2 -6732.143} C_VEL
LIN {X 0,Y 481.359,Z 252.722,A -85,B 0,C 180,E1 -6734.764,E2 -6734.764} C_VEL
LIN {X 0,Y 481.56,Z 247.616,A -85,B 0,C 180,E1 -6738.211,E2 -6738.211} C_VEL
LIN {X 0,Y 481.578,Z 243.927,A -85,B 0,C 180,E1 -6740.763,E2 -6740.763} C_VEL
LIN {X 0,Y 481.659,Z 243.486,A -85,B 0,C 180,E1 -6741.61,E2 -6741.61} C_VEL
LIN {X 0,Y 481.804,Z 243.471,A -85,B 0,C 180,E1 -6744.14,E2 -6744.14} C_VEL
LIN {X 0,Y 481.917,Z 243.456,A -85,B 0,C 180,E1 -6747.493,E2 -6747.493} C_VEL
LIN {X 0,Y 481.929,Z 243.456,A -85,B 0,C 180,E1 -6750,E2 -6750} C_VEL
LIN {X 0,Y 481.92,Z 243.457,A -85,B 0,C 180,E1 -6752.508,E2 -6752.508} C_VEL
LIN {X 0,Y 481.807,Z 243.472,A -85,B 0,C 180,E1 -6755.861,E2 -6755.861} C_VEL
LIN {X 0,Y 481.753,Z 243.478,A -85,B 0,C 180,E1 -6758.388,E2 -6758.388} C_VEL
LIN {X 0,Y 481.785,Z 243.475,A -85,B 0,C 180,E1 -6761.784,E2 -6761.784} C_VEL
LIN {X 0,Y 481.731,Z 243.48,A -85,B 0,C 180,E1 -6765.224,E2 -6765.224} C_VEL
LIN {X 0,Y 481.701,Z 243.484,A -85,B 0,C 180,E1 -6768.722,E2 -6768.722} C_VEL
LIN {X 0,Y 481.661,Z 243.489,A -85,B 0,C 180,E1 -6771.394,E2 -6771.394} C_VEL
LIN {X 0,Y 481.672,Z 243.487,A -85,B 0,C 180,E1 -6774.113,E2 -6774.113} C_VEL
LIN {X 0,Y 481.741,Z 243.478,A -85,B 0,C 180,E1 -6777.141,E2 -6777.141} C_VEL
LIN {X 0,Y 481.677,Z 243.488,A -85,B 0,C 180,E1 -6779.741,E2 -6779.741} C_VEL
LIN {X 0,Y 481.662,Z 243.487,A -85,B 0,C 180,E1 -6782.674,E2 -6782.674} C_VEL
LIN {X 0,Y 481.631,Z 243.494,A -85,B 0,C 180,E1 -6785.709,E2 -6785.709} C_VEL
LIN {X 0,Y 481.708,Z 243.485,A -85,B 0,C 180,E1 -6789.355,E2 -6789.355} C_VEL
LIN {X 0,Y 481.663,Z 243.487,A -85,B 0,C 180,E1 -6792.158,E2 -6792.158} C_VEL
LIN {X 0,Y 481.649,Z 243.489,A -85,B 0,C 180,E1 -6794.458,E2 -6794.458} C_VEL
LIN {X 0,Y 481.678,Z 243.487,A -85,B 0,C 180,E1 -6796.846,E2 -6796.846} C_VEL
LIN {X 0,Y 481.681,Z 243.486,A -85,B 0,C 180,E1 -6800.062,E2 -6800.062} C_VEL
LIN {X 0,Y 481.619,Z 243.495,A -85,B 0,C 180,E1 -6803.254,E2 -6803.254} C_VEL
LIN {X 0,Y 481.699,Z 243.484,A -85,B 0,C 180,E1 -6806.331,E2 -6806.331} C_VEL
LIN {X 0,Y 481.648,Z 243.492,A -85,B 0,C 180,E1 -6809.416,E2 -6809.416} C_VEL
LIN {X 0,Y 481.693,Z 243.485,A -85,B 0,C 180,E1 -6812.169,E2 -6812.169} C_VEL
LIN {X 0,Y 481.709,Z 243.483,A -85,B 0,C 180,E1 -6814.971,E2 -6814.971} C_VEL
LIN {X 0,Y 481.643,Z 243.49,A -85,B 0,C 180,E1 -6817.706,E2 -6817.706} C_VEL
LIN {X 0,Y 481.699,Z 243.485,A -85,B 0,C 180,E1 -6820.394,E2 -6820.394} C_VEL
LIN {X 0,Y 481.683,Z 243.486,A -85,B 0,C 180,E1 -6823.035,E2 -6823.035} C_VEL
LIN {X 0,Y 481.68,Z 243.485,A -85,B 0,C 180,E1 -6825.64,E2 -6825.64} C_VEL
LIN {X 0,Y 481.744,Z 243.478,A -85,B 0,C 180,E1 -6828.216,E2 -6828.216} C_VEL
LIN {X 0,Y 481.756,Z 243.476,A -85,B 0,C 180,E1 -6831.613,E2 -6831.613} C_VEL
LIN {X 0,Y 481.808,Z 243.471,A -85,B 0,C 180,E1 -6834.141,E2 -6834.141} C_VEL
LIN {X 0,Y 481.921,Z 243.456,A -85,B 0,C 180,E1 -6837.494,E2 -6837.494} C_VEL
LIN {X 0,Y 481.9,Z 243.459,A -85,B 0,C 180,E1 -6840.837,E2 -6840.837} C_VEL
LIN {X 0,Y 481.923,Z 243.456,A -85,B 0,C 180,E1 -6842.508,E2 -6842.508} C_VEL
LIN {X 0,Y 481.81,Z 243.471,A -85,B 0,C 180,E1 -6845.861,E2 -6845.861} C_VEL
LIN {X 0,Y 481.757,Z 243.476,A -85,B 0,C 180,E1 -6848.389,E2 -6848.389} C_VEL
LIN {X 0,Y 481.79,Z 243.474,A -85,B 0,C 180,E1 -6851.785,E2 -6851.785} C_VEL
LIN {X 0,Y 481.738,Z 243.479,A -85,B 0,C 180,E1 -6855.225,E2 -6855.225} C_VEL
LIN {X 0,Y 481.708,Z 243.483,A -85,B 0,C 180,E1 -6858.723,E2 -6858.723} C_VEL
LIN {X 0,Y 481.642,Z 243.493,A -85,B 0,C 180,E1 -6861.396,E2 -6861.396} C_VEL
LIN {X 0,Y 481.673,Z 243.486,A -85,B 0,C 180,E1 -6864.114,E2 -6864.114} C_VEL
LIN {X 0,Y 481.744,Z 243.479,A -85,B 0,C 180,E1 -6867.14,E2 -6867.14} C_VEL
LIN {X 0,Y 481.676,Z 243.488,A -85,B 0,C 180,E1 -6869.742,E2 -6869.742} C_VEL
LIN {X 0,Y 481.668,Z 243.486,A -85,B 0,C 180,E1 -6872.675,E2 -6872.675} C_VEL
LIN {X 0,Y 481.639,Z 243.492,A -85,B 0,C 180,E1 -6875.71,E2 -6875.71} C_VEL
LIN {X 0,Y 481.67,Z 243.487,A -85,B 0,C 180,E1 -6878.86,E2 -6878.86} C_VEL
LIN {X 0,Y 481.652,Z 243.488,A -85,B 0,C 180,E1 -6881.914,E2 -6881.914} C_VEL
LIN {X 0,Y 481.654,Z 243.489,A -85,B 0,C 180,E1 -6884.459,E2 -6884.459} C_VEL
LIN {X 0,Y 481.648,Z 243.491,A -85,B 0,C 180,E1 -6887.84,E2 -6887.84} C_VEL
LIN {X 0,Y 481.698,Z 243.484,A -85,B 0,C 180,E1 -6891.144,E2 -6891.144} C_VEL
LIN {X 0,Y 481.71,Z 243.519,A -85,B 0,C 180,E1 -6891.366,E2 -6891.366} C_VEL
LIN {X 0,Y 482.462,Z 248.541,A -85,B 0,C 180,E1 -6893.846,E2 -6893.846} C_VEL
LIN {X 0,Y 482.455,Z 254,A -85,B 0,C 180,E1 -6896.39,E2 -6896.39} C_VEL
LIN {X 0,Y 482.159,Z 260.578,A -85,B 0,C 180,E1 -6899.326,E2 -6899.326} C_VEL
LIN {X 0,Y 481.841,Z 267.172,A -85,B 0,C 180,E1 -6902.177,E2 -6902.177} C_VEL
LIN {X 0,Y 481.655,Z 273.771,A -85,B 0,C 180,E1 -6904.967,E2 -6904.967} C_VEL
LIN {X 0,Y 481.453,Z 281.503,A -85,B 0,C 180,E1 -6908.147,E2 -6908.147} C_VEL
LIN {X 0,Y 481.276,Z 289.252,A -85,B 0,C 180,E1 -6911.261,E2 -6911.261} C_VEL
LIN {X 0,Y 481.12,Z 297.708,A -85,B 0,C 180,E1 -6914.603,E2 -6914.603} C_VEL
LIN {X 0,Y 481.105,Z 299.094,A -85,B 0,C 180,E1 -6915.08,E2 -6915.08} C_VEL
LIN {X 0,Y 483.2,Z 312.491,A -85,B 0,C 180,E1 -6915.497,E2 -6915.497} C_VEL
LIN {X 0,Y 483.787,Z 317.73,A -85,B 0,C 180,E1 -6915.702,E2 -6915.702} C_VEL
LIN {X 0,Y 483.446,Z 329.427,A -85,B 0,C 180,E1 -6916.229,E2 -6916.229} C_VEL
LIN {X 0,Y 482.991,Z 340.671,A -85,B 0,C 180,E1 -6916.891,E2 -6916.891} C_VEL
LIN {X 0,Y 482.515,Z 351.709,A -85,B 0,C 180,E1 -6917.714,E2 -6917.714} C_VEL
LIN {X 0,Y 482.211,Z 361.818,A -85,B 0,C 180,E1 -6918.653,E2 -6918.653} C_VEL
LIN {X 0,Y 481.745,Z 371.039,A -85,B 0,C 180,E1 -6919.705,E2 -6919.705} C_VEL
LIN {X 0,Y 481.416,Z 380.017,A -85,B 0,C 180,E1 -6920.971,E2 -6920.971} C_VEL
LIN {X 0,Y 481.153,Z 387.248,A -85,B 0,C 180,E1 -6922.235,E2 -6922.235} C_VEL
LIN {X 0,Y 480.97,Z 393.15,A -85,B 0,C 180,E1 -6923.531,E2 -6923.531} C_VEL
LIN {X 0,Y 480.898,Z 398.189,A -85,B 0,C 180,E1 -6924.969,E2 -6924.969} C_VEL
LIN {X 0,Y 480.828,Z 400.49,A -85,B 0,C 180,E1 -6925.809,E2 -6925.809} C_VEL
LIN {X 0,Y 480.889,Z 402.36,A -85,B 0,C 180,E1 -6926.649,E2 -6926.649} C_VEL
LIN {X 0,Y 480.824,Z 403.758,A -85,B 0,C 180,E1 -6927.487,E2 -6927.487} C_VEL
LIN {X 0,Y 480.793,Z 404.753,A -85,B 0,C 180,E1 -6928.325,E2 -6928.325} C_VEL
LIN {X 0,Y 480.76,Z 405.359,A -85,B 0,C 180,E1 -6929.162,E2 -6929.162} C_VEL
LIN {X 0,Y 480.743,Z 405.571,A -85,B 0,C 180,E1 -6930,E2 -6930} C_VEL
LIN {X 0,Y 480.76,Z 405.349,A -85,B 0,C 180,E1 -6930.837,E2 -6930.837} C_VEL
LIN {X 0,Y 480.793,Z 404.734,A -85,B 0,C 180,E1 -6931.675,E2 -6931.675} C_VEL
LIN {X 0,Y 480.824,Z 403.729,A -85,B 0,C 180,E1 -6932.513,E2 -6932.513} C_VEL
LIN {X 0,Y 480.889,Z 402.321,A -85,B 0,C 180,E1 -6933.351,E2 -6933.351} C_VEL
LIN {X 0,Y 480.839,Z 399.36,A -85,B 0,C 180,E1 -6934.611,E2 -6934.611} C_VEL
LIN {X 0,Y 480.93,Z 395.356,A -85,B 0,C 180,E1 -6935.871,E2 -6935.871} C_VEL
LIN {X 0,Y 481.113,Z 389.199,A -85,B 0,C 180,E1 -6937.343,E2 -6937.343} C_VEL
LIN {X 0,Y 481.325,Z 382.475,A -85,B 0,C 180,E1 -6938.607,E2 -6938.607} C_VEL
LIN {X 0,Y 481.64,Z 374.137,A -85,B 0,C 180,E1 -6939.872,E2 -6939.872} C_VEL
LIN {X 0,Y 482.018,Z 365.582,A -85,B 0,C 180,E1 -6940.926,E2 -6940.926} C_VEL
LIN {X 0,Y 482.44,Z 355.111,A -85,B 0,C 180,E1 -6941.973,E2 -6941.973} C_VEL
LIN {X 0,Y 482.838,Z 343.6,A -85,B 0,C 180,E1 -6942.899,E2 -6942.899} C_VEL
LIN {X 0,Y 483.346,Z 331.223,A -85,B 0,C 180,E1 -6943.667,E2 -6943.667} C_VEL
LIN {X 0,Y 483.743,Z 318.86,A -85,B 0,C 180,E1 -6944.245,E2 -6944.245} C_VEL
LIN {X 0,Y 483.388,Z 313.873,A -85,B 0,C 180,E1 -6944.444,E2 -6944.444} C_VEL
LIN {X 0,Y 481.397,Z 300.932,A -85,B 0,C 180,E1 -6944.876,E2 -6944.876} C_VEL
LIN {X 0,Y 481.063,Z 298.582,A -85,B 0,C 180,E1 -6944.948,E2 -6944.948} C_VEL
LIN {X 0,Y 481.176,Z 291.132,A -85,B 0,C 180,E1 -6947.861,E2 -6947.861} C_VEL
LIN {X 0,Y 481.348,Z 283.609,A -85,B 0,C 180,E1 -6950.86,E2 -6950.86} C_VEL
LIN {X 0,Y 481.529,Z 276.735,A -85,B 0,C 180,E1 -6953.663,E2 -6953.663} C_VEL
LIN {X 0,Y 481.72,Z 270.159,A -85,B 0,C 180,E1 -6956.421,E2 -6956.421} C_VEL
LIN {X 0,Y 482.11,Z 261.512,A -85,B 0,C 180,E1 -6960.193,E2 -6960.193} C_VEL
LIN {X 0,Y 482.352,Z 255.118,A -85,B 0,C 180,E1 -6963.118,E2 -6963.118} C_VEL
LIN {X 0,Y 482.548,Z 249.896,A -85,B 0,C 180,E1 -6965.631,E2 -6965.631} C_VEL
LIN {X 0,Y 482.108,Z 245.79,A -85,B 0,C 180,E1 -6967.752,E2 -6967.752} C_VEL
LIN {X 0,Y 481.673,Z 243.49,A -85,B 0,C 180,E1 -6969.103,E2 -6969.103} C_VEL
LIN {X 0,Y 481.653,Z 243.492,A -85,B 0,C 180,E1 -6972.159,E2 -6972.159} C_VEL
LIN {X 0,Y 481.658,Z 243.492,A -85,B 0,C 180,E1 -6975.542,E2 -6975.542} C_VEL
LIN {X 0,Y 481.666,Z 243.49,A -85,B 0,C 180,E1 -6978.958,E2 -6978.958} C_VEL
LIN {X 0,Y 481.695,Z 243.486,A -85,B 0,C 180,E1 -6981.142,E2 -6981.142} C_VEL
LIN {X 0,Y 481.666,Z 243.49,A -85,B 0,C 180,E1 -6984.794,E2 -6984.794} C_VEL
LIN {X 0,Y 481.67,Z 243.488,A -85,B 0,C 180,E1 -6987.325,E2 -6987.325} C_VEL
LIN {X 0,Y 481.684,Z 243.486,A -85,B 0,C 180,E1 -6990.258,E2 -6990.258} C_VEL
LIN {X 0,Y 481.741,Z 243.479,A -85,B 0,C 180,E1 -6993.111,E2 -6993.111} C_VEL
LIN {X 0,Y 481.672,Z 243.489,A -85,B 0,C 180,E1 -6995.886,E2 -6995.886} C_VEL
LIN {X 0,Y 481.697,Z 243.486,A -85,B 0,C 180,E1 -6999.026,E2 -6999.026} C_VEL
LIN {X 0,Y 481.701,Z 243.486,A -85,B 0,C 180,E1 -7002.157,E2 -7002.157} C_VEL
LIN {X 0,Y 481.736,Z 243.48,A -85,B 0,C 180,E1 -7004.775,E2 -7004.775} C_VEL
LIN {X 0,Y 481.746,Z 243.48,A -85,B 0,C 180,E1 -7008.214,E2 -7008.214} C_VEL
LIN {X 0,Y 481.757,Z 243.478,A -85,B 0,C 180,E1 -7011.611,E2 -7011.611} C_VEL
LIN {X 0,Y 481.81,Z 243.471,A -85,B 0,C 180,E1 -7014.139,E2 -7014.139} C_VEL
LIN {X 0,Y 481.92,Z 243.459,A -85,B 0,C 180,E1 -7017.492,E2 -7017.492} C_VEL
LIN {X 0,Y 481.897,Z 243.46,A -85,B 0,C 180,E1 -7020.835,E2 -7020.835} C_VEL
LIN {X 0,Y 481.921,Z 243.459,A -85,B 0,C 180,E1 -7022.506,E2 -7022.506} C_VEL
LIN {X 0,Y 481.808,Z 243.472,A -85,B 0,C 180,E1 -7025.859,E2 -7025.859} C_VEL
LIN {X 0,Y 481.752,Z 243.479,A -85,B 0,C 180,E1 -7028.387,E2 -7028.387} C_VEL
LIN {X 0,Y 481.633,Z 243.496,A -85,B 0,C 180,E1 -7030.084,E2 -7030.084} C_VEL
LIN {X 0,Y 481.727,Z 246.185,A -85,B 0,C 180,E1 -7032.19,E2 -7032.19} C_VEL
LIN {X 0,Y 481.54,Z 250.991,A -85,B 0,C 180,E1 -7035.584,E2 -7035.584} C_VEL
LIN {X 0,Y 481.389,Z 255.564,A -85,B 0,C 180,E1 -7038.734,E2 -7038.734} C_VEL
LIN {X 0,Y 481.262,Z 259.54,A -85,B 0,C 180,E1 -7041.411,E2 -7041.411} C_VEL
LIN {X 0,Y 481.175,Z 263.677,A -85,B 0,C 180,E1 -7044.139,E2 -7044.139} C_VEL
LIN {X 0,Y 481.093,Z 268.06,A -85,B 0,C 180,E1 -7046.989,E2 -7046.989} C_VEL
LIN {X 0,Y 480.924,Z 273.486,A -85,B 0,C 180,E1 -7050.438,E2 -7050.438} C_VEL
LIN {X 0,Y 480.945,Z 274.567,A -85,B 0,C 180,E1 -7051.125,E2 -7051.125} C_VEL
LIN {X 0,Y 483.941,Z 289.475,A -85,B 0,C 180,E1 -7051.68,E2 -7051.68} C_VEL
LIN {X 0,Y 483.655,Z 302.051,A -85,B 0,C 180,E1 -7052.226,E2 -7052.226} C_VEL
LIN {X 0,Y 483.222,Z 313.994,A -85,B 0,C 180,E1 -7052.926,E2 -7052.926} C_VEL
LIN {X 0,Y 482.807,Z 324.948,A -85,B 0,C 180,E1 -7053.747,E2 -7053.747} C_VEL
LIN {X 0,Y 482.365,Z 335.567,A -85,B 0,C 180,E1 -7054.74,E2 -7054.74} C_VEL
LIN {X 0,Y 481.948,Z 344.777,A -85,B 0,C 180,E1 -7055.81,E2 -7055.81} C_VEL
LIN {X 0,Y 481.591,Z 353.19,A -85,B 0,C 180,E1 -7057.01,E2 -7057.01} C_VEL
LIN {X 0,Y 481.274,Z 360.997,A -85,B 0,C 180,E1 -7058.401,E2 -7058.401} C_VEL
LIN {X 0,Y 481.075,Z 366.36,A -85,B 0,C 180,E1 -7059.607,E2 -7059.607} C_VEL
LIN {X 0,Y 480.948,Z 371.513,A -85,B 0,C 180,E1 -7061.114,E2 -7061.114} C_VEL
LIN {X 0,Y 480.819,Z 374.411,A -85,B 0,C 180,E1 -7062.248,E2 -7062.248} C_VEL
LIN {X 0,Y 480.724,Z 376.553,A -85,B 0,C 180,E1 -7063.401,E2 -7063.401} C_VEL
LIN {X 0,Y 480.748,Z 377.888,A -85,B 0,C 180,E1 -7064.562,E2 -7064.562} C_VEL
LIN {X 0,Y 480.728,Z 378.464,A -85,B 0,C 180,E1 -7065.752,E2 -7065.752} C_VEL
LIN {X 0,Y 480.672,Z 378.239,A -85,B 0,C 180,E1 -7066.973,E2 -7066.973} C_VEL
LIN {X 0,Y 480.744,Z 377.161,A -85,B 0,C 180,E1 -7068.206,E2 -7068.206} C_VEL
LIN {X 0,Y 480.797,Z 375.142,A -85,B 0,C 180,E1 -7069.471,E2 -7069.471} C_VEL
LIN {X 0,Y 480.919,Z 371.168,A -85,B 0,C 180,E1 -7071.07,E2 -7071.07} C_VEL
LIN {X 0,Y 481.064,Z 366.522,A -85,B 0,C 180,E1 -7072.416,E2 -7072.416} C_VEL
LIN {X 0,Y 481.297,Z 360.048,A -85,B 0,C 180,E1 -7073.854,E2 -7073.854} C_VEL
LIN {X 0,Y 481.547,Z 353.147,A -85,B 0,C 180,E1 -7075.066,E2 -7075.066} C_VEL
LIN {X 0,Y 481.944,Z 344.08,A -85,B 0,C 180,E1 -7076.349,E2 -7076.349} C_VEL
LIN {X 0,Y 482.309,Z 335.155,A -85,B 0,C 180,E1 -7077.375,E2 -7077.375} C_VEL
LIN {X 0,Y 482.732,Z 324.155,A -85,B 0,C 180,E1 -7078.392,E2 -7078.392} C_VEL
LIN {X 0,Y 482.962,Z 318.698,A -85,B 0,C 180,E1 -7078.818,E2 -7078.818} C_VEL
LIN {X 0,Y 482.417,Z 315.395,A -85,B 0,C 180,E1 -7079.077,E2 -7079.077} C_VEL
LIN {X 0,Y 479.781,Z 310.258,A -85,B 0,C 180,E1 -7079.503,E2 -7079.503} C_VEL
LIN {X 0,Y 477.177,Z 304.955,A -85,B 0,C 180,E1 -7079.894,E2 -7079.894} C_VEL
LIN {X 0,Y 476.666,Z 301.382,A -85,B 0,C 180,E1 -7080.094,E2 -7080.094} C_VEL
LIN {X 0,Y 476.914,Z 290.169,A -85,B 0,C 180,E1 -7080.589,E2 -7080.589} C_VEL
LIN {X 0,Y 474.456,Z 277.701,A -85,B 0,C 180,E1 -7081.06,E2 -7081.06} C_VEL
LIN {X 0,Y 473.838,Z 274.397,A -85,B 0,C 180,E1 -7081.177,E2 -7081.177} C_VEL
LIN {X 0,Y 473.876,Z 270.599,A -85,B 0,C 180,E1 -7083.582,E2 -7083.582} C_VEL
LIN {X 0,Y 474.004,Z 265.545,A -85,B 0,C 180,E1 -7086.815,E2 -7086.815} C_VEL
LIN {X 0,Y 474.125,Z 260.547,A -85,B 0,C 180,E1 -7090.067,E2 -7090.067} C_VEL
LIN {X 0,Y 474.207,Z 256.483,A -85,B 0,C 180,E1 -7092.758,E2 -7092.758} C_VEL
LIN {X 0,Y 474.303,Z 252.542,A -85,B 0,C 180,E1 -7095.411,E2 -7095.411} C_VEL
LIN {X 0,Y 474.51,Z 248.693,A -85,B 0,C 180,E1 -7098.033,E2 -7098.033} C_VEL
LIN {X 0,Y 474.522,Z 244.986,A -85,B 0,C 180,E1 -7100.624,E2 -7100.624} C_VEL
LIN {X 0,Y 474.605,Z 244.365,A -85,B 0,C 180,E1 -7101.485,E2 -7101.485} C_VEL
LIN {X 0,Y 474.765,Z 244.347,A -85,B 0,C 180,E1 -7104.052,E2 -7104.052} C_VEL
LIN {X 0,Y 474.884,Z 244.332,A -85,B 0,C 180,E1 -7107.456,E2 -7107.456} C_VEL
LIN {X 0,Y 474.9,Z 244.331,A -85,B 0,C 180,E1 -7110,E2 -7110} C_VEL
LIN {X 0,Y 474.886,Z 244.333,A -85,B 0,C 180,E1 -7112.545,E2 -7112.545} C_VEL
LIN {X 0,Y 474.769,Z 244.348,A -85,B 0,C 180,E1 -7115.948,E2 -7115.948} C_VEL
LIN {X 0,Y 474.719,Z 244.354,A -85,B 0,C 180,E1 -7118.514,E2 -7118.514} C_VEL
LIN {X 0,Y 474.729,Z 244.353,A -85,B 0,C 180,E1 -7121.962,E2 -7121.962} C_VEL
LIN {X 0,Y 474.691,Z 244.357,A -85,B 0,C 180,E1 -7125.777,E2 -7125.777} C_VEL
LIN {X 0,Y 474.655,Z 244.361,A -85,B 0,C 180,E1 -7129.01,E2 -7129.01} C_VEL
LIN {X 0,Y 474.626,Z 244.365,A -85,B 0,C 180,E1 -7131.727,E2 -7131.727} C_VEL
LIN {X 0,Y 474.651,Z 244.363,A -85,B 0,C 180,E1 -7134.493,E2 -7134.493} C_VEL
LIN {X 0,Y 474.688,Z 244.358,A -85,B 0,C 180,E1 -7137.339,E2 -7137.339} C_VEL
LIN {X 0,Y 474.599,Z 244.368,A -85,B 0,C 180,E1 -7140.812,E2 -7140.812} C_VEL
LIN {X 0,Y 474.627,Z 244.365,A -85,B 0,C 180,E1 -7143.984,E2 -7143.984} C_VEL
LIN {X 0,Y 474.565,Z 244.373,A -85,B 0,C 180,E1 -7146.9,E2 -7146.9} C_VEL
LIN {X 0,Y 474.643,Z 244.363,A -85,B 0,C 180,E1 -7149.652,E2 -7149.652} C_VEL
LIN {X 0,Y 474.641,Z 244.364,A -85,B 0,C 180,E1 -7152.93,E2 -7152.93} C_VEL
LIN {X 0,Y 474.607,Z 244.367,A -85,B 0,C 180,E1 -7155.897,E2 -7155.897} C_VEL
LIN {X 0,Y 474.634,Z 244.366,A -85,B 0,C 180,E1 -7159.039,E2 -7159.039} C_VEL
LIN {X 0,Y 474.609,Z 244.367,A -85,B 0,C 180,E1 -7161.703,E2 -7161.703} C_VEL
LIN {X 0,Y 474.619,Z 244.366,A -85,B 0,C 180,E1 -7164.727,E2 -7164.727} C_VEL
LIN {X 0,Y 474.627,Z 244.364,A -85,B 0,C 180,E1 -7167.789,E2 -7167.789} C_VEL
LIN {X 0,Y 474.622,Z 244.368,A -85,B 0,C 180,E1 -7170.883,E2 -7170.883} C_VEL
LIN {X 0,Y 474.656,Z 244.359,A -85,B 0,C 180,E1 -7173.63,E2 -7173.63} C_VEL
LIN {X 0,Y 474.626,Z 244.366,A -85,B 0,C 180,E1 -7176.642,E2 -7176.642} C_VEL
LIN {X 0,Y 474.647,Z 244.361,A -85,B 0,C 180,E1 -7180.091,E2 -7180.091} C_VEL
LIN {X 0,Y 474.642,Z 244.365,A -85,B 0,C 180,E1 -7182.775,E2 -7182.775} C_VEL
LIN {X 0,Y 474.639,Z 244.362,A -85,B 0,C 180,E1 -7185.422,E2 -7185.422} C_VEL
LIN {X 0,Y 474.697,Z 244.356,A -85,B 0,C 180,E1 -7188.039,E2 -7188.039} C_VEL
LIN {X 0,Y 474.721,Z 244.352,A -85,B 0,C 180,E1 -7191.487,E2 -7191.487} C_VEL
LIN {X 0,Y 474.771,Z 244.347,A -85,B 0,C 180,E1 -7194.053,E2 -7194.053} C_VEL
LIN {X 0,Y 474.887,Z 244.332,A -85,B 0,C 180,E1 -7197.456,E2 -7197.456} C_VEL
LIN {X 0,Y 474.852,Z 244.337,A -85,B 0,C 180,E1 -7200.849,E2 -7200.849} C_VEL
LIN {X 0,Y 474.889,Z 244.332,A -85,B 0,C 180,E1 -7202.546,E2 -7202.546} C_VEL
LIN {X 0,Y 474.773,Z 244.348,A -85,B 0,C 180,E1 -7205.949,E2 -7205.949} C_VEL
LIN {X 0,Y 474.722,Z 244.352,A -85,B 0,C 180,E1 -7208.515,E2 -7208.515} C_VEL
LIN {X 0,Y 474.734,Z 244.352,A -85,B 0,C 180,E1 -7211.963,E2 -7211.963} C_VEL
LIN {X 0,Y 474.676,Z 244.359,A -85,B 0,C 180,E1 -7215.769,E2 -7215.769} C_VEL
LIN {X 0,Y 474.661,Z 244.361,A -85,B 0,C 180,E1 -7219.011,E2 -7219.011} C_VEL
LIN {X 0,Y 474.585,Z 244.37,A -85,B 0,C 180,E1 -7221.73,E2 -7221.73} C_VEL
LIN {X 0,Y 474.656,Z 244.361,A -85,B 0,C 180,E1 -7224.494,E2 -7224.494} C_VEL
LIN {X 0,Y 474.678,Z 244.361,A -85,B 0,C 180,E1 -7227.335,E2 -7227.335} C_VEL
LIN {X 0,Y 474.602,Z 244.367,A -85,B 0,C 180,E1 -7230.231,E2 -7230.231} C_VEL
LIN {X 0,Y 474.631,Z 244.366,A -85,B 0,C 180,E1 -7233.222,E2 -7233.222} C_VEL
LIN {X 0,Y 474.59,Z 244.367,A -85,B 0,C 180,E1 -7236.324,E2 -7236.324} C_VEL
LIN {X 0,Y 474.627,Z 244.364,A -85,B 0,C 180,E1 -7239.649,E2 -7239.649} C_VEL
LIN {X 0,Y 474.606,Z 244.37,A -85,B 0,C 180,E1 -7242.936,E2 -7242.936} C_VEL
LIN {X 0,Y 474.606,Z 244.366,A -85,B 0,C 180,E1 -7245.896,E2 -7245.896} C_VEL
LIN {X 0,Y 474.629,Z 244.365,A -85,B 0,C 180,E1 -7249.042,E2 -7249.042} C_VEL
LIN {X 0,Y 474.687,Z 244.453,A -85,B 0,C 180,E1 -7251.211,E2 -7251.211} C_VEL
LIN {X 0,Y 475.454,Z 249.518,A -85,B 0,C 180,E1 -7253.754,E2 -7253.754} C_VEL
LIN {X 0,Y 475.484,Z 253.965,A -85,B 0,C 180,E1 -7255.866,E2 -7255.866} C_VEL
LIN {X 0,Y 475.152,Z 261.022,A -85,B 0,C 180,E1 -7259.081,E2 -7259.081} C_VEL
LIN {X 0,Y 474.847,Z 267.035,A -85,B 0,C 180,E1 -7261.731,E2 -7261.731} C_VEL
LIN {X 0,Y 474.608,Z 274.751,A -85,B 0,C 180,E1 -7265.043,E2 -7265.043} C_VEL
LIN {X 0,Y 474.399,Z 282.453,A -85,B 0,C 180,E1 -7268.262,E2 -7268.262} C_VEL
LIN {X 0,Y 474.207,Z 290.479,A -85,B 0,C 180,E1 -7271.536,E2 -7271.536} C_VEL
LIN {X 0,Y 474.056,Z 298.756,A -85,B 0,C 180,E1 -7274.853,E2 -7274.853} C_VEL
LIN {X 0,Y 476.195,Z 312.542,A -85,B 0,C 180,E1 -7275.292,E2 -7275.292} C_VEL
LIN {X 0,Y 476.84,Z 318.724,A -85,B 0,C 180,E1 -7275.544,E2 -7275.544} C_VEL
LIN {X 0,Y 476.437,Z 331.125,A -85,B 0,C 180,E1 -7276.131,E2 -7276.131} C_VEL
LIN {X 0,Y 475.943,Z 343.089,A -85,B 0,C 180,E1 -7276.878,E2 -7276.878} C_VEL
LIN {X 0,Y 475.493,Z 354.208,A -85,B 0,C 180,E1 -7277.772,E2 -7277.772} C_VEL
LIN {X 0,Y 475.144,Z 363.552,A -85,B 0,C 180,E1 -7278.698,E2 -7278.698} C_VEL
LIN {X 0,Y 474.626,Z 372.445,A -85,B 0,C 180,E1 -7279.765,E2 -7279.765} C_VEL
LIN {X 0,Y 474.313,Z 381.135,A -85,B 0,C 180,E1 -7281.05,E2 -7281.05} C_VEL
LIN {X 0,Y 474.046,Z 388.068,A -85,B 0,C 180,E1 -7282.332,E2 -7282.332} C_VEL
LIN {X 0,Y 473.875,Z 393.397,A -85,B 0,C 180,E1 -7283.554,E2 -7283.554} C_VEL
LIN {X 0,Y 473.829,Z 397.983,A -85,B 0,C 180,E1 -7284.894,E2 -7284.894} C_VEL
LIN {X 0,Y 473.735,Z 400.286,A -85,B 0,C 180,E1 -7285.746,E2 -7285.746} C_VEL
LIN {X 0,Y 473.796,Z 402.158,A -85,B 0,C 180,E1 -7286.598,E2 -7286.598} C_VEL
LIN {X 0,Y 473.742,Z 403.558,A -85,B 0,C 180,E1 -7287.449,E2 -7287.449} C_VEL
LIN {X 0,Y 473.689,Z 405.159,A -85,B 0,C 180,E1 -7289.15,E2 -7289.15} C_VEL
LIN {X 0,Y 473.67,Z 405.372,A -85,B 0,C 180,E1 -7290,E2 -7290} C_VEL
LIN {X 0,Y 473.689,Z 405.15,A -85,B 0,C 180,E1 -7290.85,E2 -7290.85} C_VEL
LIN {X 0,Y 473.742,Z 403.528,A -85,B 0,C 180,E1 -7292.551,E2 -7292.551} C_VEL
LIN {X 0,Y 473.796,Z 402.118,A -85,B 0,C 180,E1 -7293.401,E2 -7293.401} C_VEL
LIN {X 0,Y 473.763,Z 399.154,A -85,B 0,C 180,E1 -7294.68,E2 -7294.68} C_VEL
LIN {X 0,Y 473.838,Z 395.146,A -85,B 0,C 180,E1 -7295.959,E2 -7295.959} C_VEL
LIN {X 0,Y 474.025,Z 388.985,A -85,B 0,C 180,E1 -7297.454,E2 -7297.454} C_VEL
LIN {X 0,Y 474.287,Z 382.26,A -85,B 0,C 180,E1 -7298.736,E2 -7298.736} C_VEL
LIN {X 0,Y 474.582,Z 373.922,A -85,B 0,C 180,E1 -7300.02,E2 -7300.02} C_VEL
LIN {X 0,Y 475.034,Z 365.37,A -85,B 0,C 180,E1 -7301.089,E2 -7301.089} C_VEL
LIN {X 0,Y 475.458,Z 355.106,A -85,B 0,C 180,E1 -7302.133,E2 -7302.133} C_VEL
LIN {X 0,Y 475.912,Z 343.395,A -85,B 0,C 180,E1 -7303.09,E2 -7303.09} C_VEL
LIN {X 0,Y 476.447,Z 331.027,A -85,B 0,C 180,E1 -7303.868,E2 -7303.868} C_VEL
LIN {X 0,Y 476.847,Z 318.684,A -85,B 0,C 180,E1 -7304.455,E2 -7304.455} C_VEL
LIN {X 0,Y 475.455,Z 307.324,A -85,B 0,C 180,E1 -7304.899,E2 -7304.899} C_VEL
LIN {X 0,Y 473.992,Z 298.374,A -85,B 0,C 180,E1 -7305.176,E2 -7305.176} C_VEL
LIN {X 0,Y 474.121,Z 290.952,A -85,B 0,C 180,E1 -7308.136,E2 -7308.136} C_VEL
LIN {X 0,Y 474.285,Z 283.89,A -85,B 0,C 180,E1 -7311.005,E2 -7311.005} C_VEL
LIN {X 0,Y 474.476,Z 276.593,A -85,B 0,C 180,E1 -7314.037,E2 -7314.037} C_VEL
LIN {X 0,Y 474.702,Z 270.051,A -85,B 0,C 180,E1 -7316.843,E2 -7316.843} C_VEL
LIN {X 0,Y 475.092,Z 262.513,A -85,B 0,C 180,E1 -7320.195,E2 -7320.195} C_VEL
LIN {X 0,Y 475.437,Z 255.144,A -85,B 0,C 180,E1 -7323.645,E2 -7323.645} C_VEL
LIN {X 0,Y 475.538,Z 249.915,A -85,B 0,C 180,E1 -7326.239,E2 -7326.239} C_VEL
LIN {X 0,Y 474.641,Z 244.366,A -85,B 0,C 180,E1 -7329.271,E2 -7329.271} C_VEL
LIN {X 0,Y 474.63,Z 244.367,A -85,B 0,C 180,E1 -7332.237,E2 -7332.237} C_VEL
LIN {X 0,Y 474.62,Z 244.367,A -85,B 0,C 180,E1 -7335.296,E2 -7335.296} C_VEL
LIN {X 0,Y 474.622,Z 244.367,A -85,B 0,C 180,E1 -7338.214,E2 -7338.214} C_VEL
LIN {X 0,Y 474.667,Z 244.363,A -85,B 0,C 180,E1 -7340.456,E2 -7340.456} C_VEL
LIN {X 0,Y 474.592,Z 244.372,A -85,B 0,C 180,E1 -7343.676,E2 -7343.676} C_VEL
LIN {X 0,Y 474.64,Z 244.365,A -85,B 0,C 180,E1 -7346.779,E2 -7346.779} C_VEL
LIN {X 0,Y 474.61,Z 244.368,A -85,B 0,C 180,E1 -7349.769,E2 -7349.769} C_VEL
LIN {X 0,Y 474.693,Z 244.357,A -85,B 0,C 180,E1 -7352.679,E2 -7352.679} C_VEL
LIN {X 0,Y 474.654,Z 244.362,A -85,B 0,C 180,E1 -7355.506,E2 -7355.506} C_VEL
LIN {X 0,Y 474.664,Z 244.362,A -85,B 0,C 180,E1 -7359.184,E2 -7359.184} C_VEL
LIN {X 0,Y 474.651,Z 244.363,A -85,B 0,C 180,E1 -7361.883,E2 -7361.883} C_VEL
LIN {X 0,Y 474.693,Z 244.357,A -85,B 0,C 180,E1 -7364.543,E2 -7364.543} C_VEL
LIN {X 0,Y 474.699,Z 244.357,A -85,B 0,C 180,E1 -7368.037,E2 -7368.037} C_VEL
LIN {X 0,Y 474.722,Z 244.355,A -85,B 0,C 180,E1 -7371.485,E2 -7371.485} C_VEL
LIN {X 0,Y 474.772,Z 244.348,A -85,B 0,C 180,E1 -7374.051,E2 -7374.051} C_VEL
LIN {X 0,Y 474.887,Z 244.334,A -85,B 0,C 180,E1 -7377.454,E2 -7377.454} C_VEL
LIN {X 0,Y 474.903,Z 244.331,A -85,B 0,C 180,E1 -7379.999,E2 -7379.999} C_VEL
LIN {X 0,Y 474.887,Z 244.335,A -85,B 0,C 180,E1 -7382.544,E2 -7382.544} C_VEL
LIN {X 0,Y 474.771,Z 244.349,A -85,B 0,C 180,E1 -7385.947,E2 -7385.947} C_VEL
LIN {X 0,Y 474.715,Z 244.356,A -85,B 0,C 180,E1 -7388.513,E2 -7388.513} C_VEL
LIN {X 0,Y 474.582,Z 244.527,A -85,B 0,C 180,E1 -7390.235,E2 -7390.235} C_VEL
LIN {X 0,Y 474.68,Z 247.255,A -85,B 0,C 180,E1 -7392.27,E2 -7392.27} C_VEL
LIN {X 0,Y 474.488,Z 252.031,A -85,B 0,C 180,E1 -7395.689,E2 -7395.689} C_VEL
LIN {X 0,Y 474.321,Z 256.793,A -85,B 0,C 180,E1 -7399.023,E2 -7399.023} C_VEL
LIN {X 0,Y 474.173,Z 260.825,A -85,B 0,C 180,E1 -7401.748,E2 -7401.748} C_VEL
LIN {X 0,Y 474.096,Z 264.98,A -85,B 0,C 180,E1 -7404.523,E2 -7404.523} C_VEL
LIN {X 0,Y 474.005,Z 269.301,A -85,B 0,C 180,E1 -7407.362,E2 -7407.362} C_VEL
LIN {X 0,Y 473.863,Z 274.804,A -85,B 0,C 180,E1 -7410.905,E2 -7410.905} C_VEL
LIN {X 0,Y 476.799,Z 288.87,A -85,B 0,C 180,E1 -7411.426,E2 -7411.426} C_VEL
LIN {X 0,Y 477.075,Z 292.873,A -85,B 0,C 180,E1 -7411.592,E2 -7411.592} C_VEL
LIN {X 0,Y 476.665,Z 305.025,A -85,B 0,C 180,E1 -7412.17,E2 -7412.17} C_VEL
LIN {X 0,Y 476.224,Z 316.468,A -85,B 0,C 180,E1 -7412.886,E2 -7412.886} C_VEL
LIN {X 0,Y 475.766,Z 327.443,A -85,B 0,C 180,E1 -7413.762,E2 -7413.762} C_VEL
LIN {X 0,Y 475.293,Z 338.104,A -85,B 0,C 180,E1 -7414.828,E2 -7414.828} C_VEL
LIN {X 0,Y 474.877,Z 346.699,A -85,B 0,C 180,E1 -7415.883,E2 -7415.883} C_VEL
LIN {X 0,Y 474.51,Z 354.86,A -85,B 0,C 180,E1 -7417.111,E2 -7417.111} C_VEL
LIN {X 0,Y 474.178,Z 362.192,A -85,B 0,C 180,E1 -7418.497,E2 -7418.497} C_VEL
LIN {X 0,Y 473.965,Z 367.983,A -85,B 0,C 180,E1 -7419.888,E2 -7419.888} C_VEL
LIN {X 0,Y 473.829,Z 372.559,A -85,B 0,C 180,E1 -7421.333,E2 -7421.333} C_VEL
LIN {X 0,Y 473.736,Z 374.465,A -85,B 0,C 180,E1 -7422.12,E2 -7422.12} C_VEL
LIN {X 0,Y 473.631,Z 376.752,A -85,B 0,C 180,E1 -7423.359,E2 -7423.359} C_VEL
LIN {X 0,Y 473.65,Z 378.132,A -85,B 0,C 180,E1 -7424.585,E2 -7424.585} C_VEL
LIN {X 0,Y 473.627,Z 378.67,A -85,B 0,C 180,E1 -7425.781,E2 -7425.781} C_VEL
LIN {X 0,Y 473.577,Z 378.459,A -85,B 0,C 180,E1 -7426.95,E2 -7426.95} C_VEL
LIN {X 0,Y 473.664,Z 377.519,A -85,B 0,C 180,E1 -7428.112,E2 -7428.112} C_VEL
LIN {X 0,Y 473.73,Z 374.73,A -85,B 0,C 180,E1 -7429.81,E2 -7429.81} C_VEL
LIN {X 0,Y 473.9,Z 370.364,A -85,B 0,C 180,E1 -7431.475,E2 -7431.475} C_VEL
LIN {X 0,Y 474.057,Z 365.126,A -85,B 0,C 180,E1 -7432.901,E2 -7432.901} C_VEL
LIN {X 0,Y 474.348,Z 358.027,A -85,B 0,C 180,E1 -7434.391,E2 -7434.391} C_VEL
LIN {X 0,Y 474.609,Z 351.408,A -85,B 0,C 180,E1 -7435.501,E2 -7435.501} C_VEL
LIN {X 0,Y 475.043,Z 342.78,A -85,B 0,C 180,E1 -7436.686,E2 -7436.686} C_VEL
LIN {X 0,Y 475.473,Z 333.225,A -85,B 0,C 180,E1 -7437.751,E2 -7437.751} C_VEL
LIN {X 0,Y 475.864,Z 322.152,A -85,B 0,C 180,E1 -7438.752,E2 -7438.752} C_VEL
LIN {X 0,Y 476.328,Z 310.363,A -85,B 0,C 180,E1 -7439.585,E2 -7439.585} C_VEL
LIN {X 0,Y 476.666,Z 301.382,A -85,B 0,C 180,E1 -7440.094,E2 -7440.094} C_VEL
LIN {X 0,Y 476.146,Z 297.818,A -85,B 0,C 180,E1 -7440.285,E2 -7440.285} C_VEL
LIN {X 0,Y 474.572,Z 294.526,A -85,B 0,C 180,E1 -7440.483,E2 -7440.483} C_VEL
LIN {X 0,Y 469.863,Z 287.086,A -85,B 0,C 180,E1 -7440.928,E2 -7440.928} C_VEL
LIN {X 0,Y 468.566,Z 283.472,A -85,B 0,C 180,E1 -7441.088,E2 -7441.088} C_VEL
LIN {X 0,Y 466.754,Z 274.576,A -85,B 0,C 180,E1 -7441.411,E2 -7441.411} C_VEL
LIN {X 0,Y 466.838,Z 269.622,A -85,B 0,C 180,E1 -7444.588,E2 -7444.588} C_VEL
LIN {X 0,Y 466.961,Z 264.521,A -85,B 0,C 180,E1 -7447.898,E2 -7447.898} C_VEL
LIN {X 0,Y 467.071,Z 260.332,A -85,B 0,C 180,E1 -7450.669,E2 -7450.669} C_VEL
LIN {X 0,Y 467.171,Z 256.279,A -85,B 0,C 180,E1 -7453.392,E2 -7453.392} C_VEL
LIN {X 0,Y 467.276,Z 252.349,A -85,B 0,C 180,E1 -7456.076,E2 -7456.076} C_VEL
LIN {X 0,Y 467.458,Z 248.521,A -85,B 0,C 180,E1 -7458.729,E2 -7458.729} C_VEL
LIN {X 0,Y 467.477,Z 246.061,A -85,B 0,C 180,E1 -7460.481,E2 -7460.481} C_VEL
LIN {X 0,Y 467.545,Z 245.245,A -85,B 0,C 180,E1 -7461.355,E2 -7461.355} C_VEL
LIN {X 0,Y 467.728,Z 245.224,A -85,B 0,C 180,E1 -7463.963,E2 -7463.963} C_VEL
LIN {X 0,Y 467.849,Z 245.208,A -85,B 0,C 180,E1 -7467.417,E2 -7467.417} C_VEL
LIN {X 0,Y 467.871,Z 245.207,A -85,B 0,C 180,E1 -7470,E2 -7470} C_VEL
LIN {X 0,Y 467.851,Z 245.209,A -85,B 0,C 180,E1 -7472.583,E2 -7472.583} C_VEL
LIN {X 0,Y 467.734,Z 245.224,A -85,B 0,C 180,E1 -7476.038,E2 -7476.038} C_VEL
LIN {X 0,Y 467.672,Z 245.231,A -85,B 0,C 180,E1 -7478.643,E2 -7478.643} C_VEL
LIN {X 0,Y 467.672,Z 245.232,A -85,B 0,C 180,E1 -7482.145,E2 -7482.145} C_VEL
LIN {X 0,Y 467.656,Z 245.233,A -85,B 0,C 180,E1 -7485.893,E2 -7485.893} C_VEL
LIN {X 0,Y 467.613,Z 245.238,A -85,B 0,C 180,E1 -7489.308,E2 -7489.308} C_VEL
LIN {X 0,Y 467.556,Z 245.246,A -85,B 0,C 180,E1 -7492.072,E2 -7492.072} C_VEL
LIN {X 0,Y 467.594,Z 245.24,A -85,B 0,C 180,E1 -7494.887,E2 -7494.887} C_VEL
LIN {X 0,Y 467.617,Z 245.238,A -85,B 0,C 180,E1 -7497.769,E2 -7497.769} C_VEL
LIN {X 0,Y 467.561,Z 245.245,A -85,B 0,C 180,E1 -7501.046,E2 -7501.046} C_VEL
LIN {X 0,Y 467.578,Z 245.244,A -85,B 0,C 180,E1 -7504.243,E2 -7504.243} C_VEL
LIN {X 0,Y 467.54,Z 245.248,A -85,B 0,C 180,E1 -7507.187,E2 -7507.187} C_VEL
LIN {X 0,Y 467.586,Z 245.242,A -85,B 0,C 180,E1 -7510.263,E2 -7510.263} C_VEL
LIN {X 0,Y 467.608,Z 245.238,A -85,B 0,C 180,E1 -7512.572,E2 -7512.572} C_VEL
LIN {X 0,Y 467.563,Z 245.244,A -85,B 0,C 180,E1 -7516.177,E2 -7516.177} C_VEL
LIN {X 0,Y 467.578,Z 245.242,A -85,B 0,C 180,E1 -7518.722,E2 -7518.722} C_VEL
LIN {X 0,Y 467.567,Z 245.245,A -85,B 0,C 180,E1 -7521.407,E2 -7521.407} C_VEL
LIN {X 0,Y 467.552,Z 245.244,A -85,B 0,C 180,E1 -7524.261,E2 -7524.261} C_VEL
LIN {X 0,Y 467.572,Z 245.245,A -85,B 0,C 180,E1 -7527.321,E2 -7527.321} C_VEL
LIN {X 0,Y 467.568,Z 245.244,A -85,B 0,C 180,E1 -7530.666,E2 -7530.666} C_VEL
LIN {X 0,Y 467.618,Z 245.239,A -85,B 0,C 180,E1 -7533.201,E2 -7533.201} C_VEL
LIN {X 0,Y 467.583,Z 245.242,A -85,B 0,C 180,E1 -7536.469,E2 -7536.469} C_VEL
LIN {X 0,Y 467.615,Z 245.236,A -85,B 0,C 180,E1 -7539.778,E2 -7539.778} C_VEL
LIN {X 0,Y 467.6,Z 245.24,A -85,B 0,C 180,E1 -7542.508,E2 -7542.508} C_VEL
LIN {X 0,Y 467.597,Z 245.241,A -85,B 0,C 180,E1 -7545.197,E2 -7545.197} C_VEL
LIN {X 0,Y 467.648,Z 245.234,A -85,B 0,C 180,E1 -7547.856,E2 -7547.856} C_VEL
LIN {X 0,Y 467.675,Z 245.23,A -85,B 0,C 180,E1 -7551.358,E2 -7551.358} C_VEL
LIN {X 0,Y 467.736,Z 245.224,A -85,B 0,C 180,E1 -7553.964,E2 -7553.964} C_VEL
LIN {X 0,Y 467.853,Z 245.208,A -85,B 0,C 180,E1 -7557.418,E2 -7557.418} C_VEL
LIN {X 0,Y 467.875,Z 245.207,A -85,B 0,C 180,E1 -7560.001,E2 -7560.001} C_VEL
LIN {X 0,Y 467.854,Z 245.208,A -85,B 0,C 180,E1 -7562.584,E2 -7562.584} C_VEL
LIN {X 0,Y 467.737,Z 245.224,A -85,B 0,C 180,E1 -7566.038,E2 -7566.038} C_VEL
LIN {X 0,Y 467.676,Z 245.23,A -85,B 0,C 180,E1 -7568.644,E2 -7568.644} C_VEL
LIN {X 0,Y 467.678,Z 245.231,A -85,B 0,C 180,E1 -7572.146,E2 -7572.146} C_VEL
LIN {X 0,Y 467.645,Z 245.235,A -85,B 0,C 180,E1 -7575.886,E2 -7575.886} C_VEL
LIN {X 0,Y 467.619,Z 245.238,A -85,B 0,C 180,E1 -7579.309,E2 -7579.309} C_VEL
LIN {X 0,Y 467.531,Z 245.25,A -85,B 0,C 180,E1 -7582.075,E2 -7582.075} C_VEL
LIN {X 0,Y 467.6,Z 245.24,A -85,B 0,C 180,E1 -7584.888,E2 -7584.888} C_VEL
LIN {X 0,Y 467.618,Z 245.238,A -85,B 0,C 180,E1 -7587.77,E2 -7587.77} C_VEL
LIN {X 0,Y 467.565,Z 245.246,A -85,B 0,C 180,E1 -7591.046,E2 -7591.046} C_VEL
LIN {X 0,Y 467.586,Z 245.241,A -85,B 0,C 180,E1 -7594.243,E2 -7594.243} C_VEL
LIN {X 0,Y 467.548,Z 245.247,A -85,B 0,C 180,E1 -7597.188,E2 -7597.188} C_VEL
LIN {X 0,Y 467.577,Z 245.242,A -85,B 0,C 180,E1 -7600.266,E2 -7600.266} C_VEL
LIN {X 0,Y 467.586,Z 245.241,A -85,B 0,C 180,E1 -7602.568,E2 -7602.568} C_VEL
LIN {X 0,Y 467.566,Z 245.246,A -85,B 0,C 180,E1 -7605.053,E2 -7605.053} C_VEL
LIN {X 0,Y 467.59,Z 245.243,A -85,B 0,C 180,E1 -7607.441,E2 -7607.441} C_VEL
LIN {X 0,Y 467.631,Z 245.342,A -85,B 0,C 180,E1 -7611.025,E2 -7611.025} C_VEL
LIN {X 0,Y 468.282,Z 249.393,A -85,B 0,C 180,E1 -7613.108,E2 -7613.108} C_VEL
LIN {X 0,Y 468.528,Z 253.77,A -85,B 0,C 180,E1 -7615.25,E2 -7615.25} C_VEL
LIN {X 0,Y 468.23,Z 260.332,A -85,B 0,C 180,E1 -7618.309,E2 -7618.309} C_VEL
LIN {X 0,Y 467.897,Z 266.913,A -85,B 0,C 180,E1 -7621.272,E2 -7621.272} C_VEL
LIN {X 0,Y 467.596,Z 274.037,A -85,B 0,C 180,E1 -7624.397,E2 -7624.397} C_VEL
LIN {X 0,Y 467.37,Z 281.195,A -85,B 0,C 180,E1 -7627.453,E2 -7627.453} C_VEL
LIN {X 0,Y 467.167,Z 288.911,A -85,B 0,C 180,E1 -7630.673,E2 -7630.673} C_VEL
LIN {X 0,Y 466.996,Z 297.746,A -85,B 0,C 180,E1 -7634.283,E2 -7634.283} C_VEL
LIN {X 0,Y 466.976,Z 298.553,A -85,B 0,C 180,E1 -7634.61,E2 -7634.61} C_VEL
LIN {X 0,Y 469.322,Z 313.762,A -85,B 0,C 180,E1 -7635.13,E2 -7635.13} C_VEL
LIN {X 0,Y 469.925,Z 319.675,A -85,B 0,C 180,E1 -7635.382,E2 -7635.382} C_VEL
LIN {X 0,Y 469.448,Z 332.779,A -85,B 0,C 180,E1 -7636.031,E2 -7636.031} C_VEL
LIN {X 0,Y 468.942,Z 344.241,A -85,B 0,C 180,E1 -7636.788,E2 -7636.788} C_VEL
LIN {X 0,Y 468.484,Z 355.185,A -85,B 0,C 180,E1 -7637.703,E2 -7637.703} C_VEL
LIN {X 0,Y 468.022,Z 365.251,A -85,B 0,C 180,E1 -7638.743,E2 -7638.743} C_VEL
LIN {X 0,Y 467.552,Z 373.813,A -85,B 0,C 180,E1 -7639.827,E2 -7639.827} C_VEL
LIN {X 0,Y 467.212,Z 382.145,A -85,B 0,C 180,E1 -7641.131,E2 -7641.131} C_VEL
LIN {X 0,Y 466.951,Z 388.862,A -85,B 0,C 180,E1 -7642.432,E2 -7642.432} C_VEL
LIN {X 0,Y 466.756,Z 395.016,A -85,B 0,C 180,E1 -7643.95,E2 -7643.95} C_VEL
LIN {X 0,Y 466.69,Z 399.007,A -85,B 0,C 180,E1 -7645.249,E2 -7645.249} C_VEL
LIN {X 0,Y 466.689,Z 401.953,A -85,B 0,C 180,E1 -7646.547,E2 -7646.547} C_VEL
LIN {X 0,Y 466.663,Z 403.356,A -85,B 0,C 180,E1 -7647.41,E2 -7647.41} C_VEL
LIN {X 0,Y 466.619,Z 404.96,A -85,B 0,C 180,E1 -7649.137,E2 -7649.137} C_VEL
LIN {X 0,Y 466.599,Z 405.173,A -85,B 0,C 180,E1 -7650,E2 -7650} C_VEL
LIN {X 0,Y 466.619,Z 404.951,A -85,B 0,C 180,E1 -7650.863,E2 -7650.863} C_VEL
LIN {X 0,Y 466.663,Z 403.328,A -85,B 0,C 180,E1 -7652.589,E2 -7652.589} C_VEL
LIN {X 0,Y 466.689,Z 401.917,A -85,B 0,C 180,E1 -7653.453,E2 -7653.453} C_VEL
LIN {X 0,Y 466.69,Z 398.953,A -85,B 0,C 180,E1 -7654.751,E2 -7654.751} C_VEL
LIN {X 0,Y 466.755,Z 394.944,A -85,B 0,C 180,E1 -7656.05,E2 -7656.05} C_VEL
LIN {X 0,Y 466.951,Z 388.782,A -85,B 0,C 180,E1 -7657.567,E2 -7657.567} C_VEL
LIN {X 0,Y 467.227,Z 382.055,A -85,B 0,C 180,E1 -7658.869,E2 -7658.869} C_VEL
LIN {X 0,Y 467.55,Z 373.714,A -85,B 0,C 180,E1 -7660.173,E2 -7660.173} C_VEL
LIN {X 0,Y 468.034,Z 365.166,A -85,B 0,C 180,E1 -7661.257,E2 -7661.257} C_VEL
LIN {X 0,Y 468.473,Z 355.12,A -85,B 0,C 180,E1 -7662.297,E2 -7662.297} C_VEL
LIN {X 0,Y 468.933,Z 344.21,A -85,B 0,C 180,E1 -7663.212,E2 -7663.212} C_VEL
LIN {X 0,Y 469.456,Z 332.82,A -85,B 0,C 180,E1 -7663.969,E2 -7663.969} C_VEL
LIN {X 0,Y 469.926,Z 319.853,A -85,B 0,C 180,E1 -7664.618,E2 -7664.618} C_VEL
LIN {X 0,Y 468.945,Z 310.494,A -85,B 0,C 180,E1 -7665.01,E2 -7665.01} C_VEL
LIN {X 0,Y 466.936,Z 298.155,A -85,B 0,C 180,E1 -7665.427,E2 -7665.427} C_VEL
LIN {X 0,Y 467.08,Z 290.423,A -85,B 0,C 180,E1 -7668.568,E2 -7668.568} C_VEL
LIN {X 0,Y 467.32,Z 281.971,A -85,B 0,C 180,E1 -7672.084,E2 -7672.084} C_VEL
LIN {X 0,Y 467.576,Z 273.77,A -85,B 0,C 180,E1 -7675.597,E2 -7675.597} C_VEL
LIN {X 0,Y 467.835,Z 266.743,A -85,B 0,C 180,E1 -7678.731,E2 -7678.731} C_VEL
